SPLINE
SPL {X  -117.172, Y  +273.562, Z    +0.000, E1   -47.526, E3 -228450.483}
SPL {X  -141.985, Y  +308.763, Z    +0.000, E1   -38.695, E3 -228517.793}
SPL {X  -151.595, Y  +331.355, Z    +0.000, E1   -30.702, E3 -228532.311}
SPL {X  -155.358, Y  +344.279, Z    +0.000, E1   -24.937, E3 -228537.500}
SPL {X  -158.582, Y  +361.322, Z    +0.000, E1   -15.773, E3 -228541.844}
SPL {X  -159.657, Y  +372.183, Z    +0.000, E1    -8.995, E3 -228543.452}
SPL {X  -159.949, Y  +378.873, Z    +0.000, E1    -4.398, E3 -228544.026}
SPL {X  -159.990, Y  +382.801, Z    +0.000, E1    -1.461, E3 -228544.200}
SPL {X  -159.990, Y  +385.055, Z    +0.000, E1    +0.429, E3 -228544.239}
SPL {X  -159.990, Y  +388.743, Z    +0.000, E1    +5.147, E3 -228544.380}
SPL {X  -159.990, Y  +393.154, Z    +0.000, E1   +11.942, E3 -228544.712}
SPL {X  -159.990, Y  +397.198, Z    +0.000, E1   +18.490, E3 -228545.209}
SPL {X  -159.990, Y  +402.771, Z    +0.000, E1   +27.045, E3 -228546.172}
SPL {X  -159.990, Y  +416.096, Z    +0.000, E1   +42.325, E3 -228549.839}
SPL {X  -159.990, Y  +469.763, Z    +0.000, E1   +60.937, E3 -228575.069}
SPL {X  -159.990, Y  +561.242, Z    +0.000, E1   +63.988, E3 -228646.017}
SPL {X  -159.990, Y  +574.019, Z    +0.000, E1   +64.020, E3 -228659.184}
SPL {X  -159.990, Y  +591.720, Z    +0.000, E1   +64.032, E3 -228677.482}
SPL {X  -159.990, Y  +605.088, Z    +0.000, E1   +63.988, E3 -228691.409}
SPL {X  -159.990, Y  +614.683, Z    +0.000, E1   +63.997, E3 -228701.304}
SPL {X  -159.990, Y  +629.274, Z    +0.000, E1   +64.033, E3 -228716.335}
SPL {X  -159.990, Y  +645.396, Z    +0.000, E1   +64.010, E3 -228733.066}
SPL {X  -159.990, Y  +656.294, Z    +0.000, E1   +63.988, E3 -228744.396}
SPL {X  -159.990, Y  +667.666, Z    +0.000, E1   +64.016, E3 -228756.087}
SPL {X  -159.767, Y  +679.937, Z    +0.000, E1   +63.968, E3 -228769.063}
SPL {X  -159.113, Y  +688.225, Z    +0.000, E1   +63.867, E3 -228778.341}
SPL {X  -158.361, Y  +694.273, Z    +0.000, E1   +63.762, E3 -228785.378}
SPL {X  -157.131, Y  +701.612, Z    +0.000, E1   +63.591, E3 -228794.251}
SPL {X  -154.918, Y  +711.464, Z    +0.000, E1   +63.294, E3 -228806.686}
SPL {X  -151.874, Y  +721.810, Z    +0.000, E1   +62.834, E3 -228820.493}
SPL {X  -148.087, Y  +732.056, Z    +0.000, E1   +62.252, E3 -228834.850}
SPL {X  -144.667, Y  +739.825, Z    +0.000, E1   +61.658, E3 -228846.239}
SPL {X  -142.263, Y  +744.698, Z    +0.000, E1   +61.245, E3 -228853.554}
SPL {X  -139.956, Y  +749.019, Z    +0.000, E1   +60.852, E3 -228860.132}
SPL {X  -136.617, Y  +754.762, Z    +0.000, E1   +60.296, E3 -228868.986}
SPL {X  -132.995, Y  +760.433, Z    +0.000, E1   +59.601, E3 -228877.950}
SPL {X  -109.949, Y  +787.724, Z    +0.000, E1   +51.944, E3 -228970.511}
ENDSPLINE

SPLINE
SPL {X  -129.366, Y  +765.635, Z    +0.000, E1   +44.361, E3 -229080.253}
SPL {X  -144.719, Y  +739.715, Z    +0.000, E1   +37.620, E3 -229107.101}
SPL {X  -154.606, Y  +712.654, Z    +0.000, E1   +26.872, E3 -229120.321}
SPL {X  -158.229, Y  +695.175, Z    +0.000, E1   +17.621, E3 -229124.807}
SPL {X  -159.735, Y  +680.532, Z    +0.000, E1    +8.352, E3 -229126.899}
SPL {X  -159.976, Y  +673.579, Z    +0.000, E1    +3.308, E3 -229127.393}
SPL {X  -159.990, Y  +669.438, Z    +0.000, E1    +0.061, E3 -229127.491}
SPL {X  -159.990, Y  +667.221, Z    +0.000, E1    -2.789, E3 -229127.534}
SPL {X  -159.990, Y  +663.611, Z    +0.000, E1    -7.967, E3 -229127.724}
SPL {X  -159.990, Y  +658.381, Z    +0.000, E1   -16.786, E3 -229128.205}
SPL {X  -159.990, Y  +651.878, Z    +0.000, E1   -27.298, E3 -229129.204}
SPL {X  -159.990, Y  +644.587, Z    +0.000, E1   -37.284, E3 -229130.787}
SPL {X  -159.990, Y  +633.621, Z    +0.000, E1   -47.309, E3 -229134.278}
SPL {X  -159.990, Y  +588.658, Z    +0.000, E1   -60.812, E3 -229156.598}
SPL {X  -159.990, Y  +495.038, Z    +0.000, E1   -63.580, E3 -229231.834}
SPL {X  -159.990, Y  +483.848, Z    +0.000, E1   -63.590, E3 -229243.619}
SPL {X  -159.990, Y  +471.874, Z    +0.000, E1   -63.586, E3 -229256.245}
SPL {X  -159.990, Y  +461.079, Z    +0.000, E1   -63.579, E3 -229267.653}
SPL {X  -159.990, Y  +450.188, Z    +0.000, E1   -63.581, E3 -229279.144}
SPL {X  -159.990, Y  +442.553, Z    +0.000, E1   -63.337, E3 -229288.967}
ENDSPLINE

SPLINE
SPL {X  -159.990, Y  +465.419, Z    +0.000, E1   -58.181, E3 -229297.813}
ENDSPLINE

SPLINE
SPL {X  -159.990, Y  +455.003, Z    +0.000, E1   -58.788, E3 -229307.351}
SPL {X  -159.990, Y  +443.180, Z    +0.000, E1   -59.522, E3 -229317.389}
SPL {X  -159.990, Y  +431.227, Z    +0.000, E1   -60.120, E3 -229328.081}
SPL {X  -159.990, Y  +413.464, Z    +0.000, E1   -61.043, E3 -229343.071}
SPL {X  -159.990, Y  +395.417, Z    +0.000, E1   -62.063, E3 -229356.514}
SPL {X  -159.983, Y  +381.042, Z    +0.000, E1   -62.802, E3 -229367.145}
SPL {X  -159.542, Y  +370.537, Z    +0.000, E1   -63.069, E3 -229376.527}
SPL {X  -158.758, Y  +362.683, Z    +0.000, E1   -62.956, E3 -229385.801}
SPL {X  -157.125, Y  +352.357, Z    +0.000, E1   -62.751, E3 -229398.534}
SPL {X  -154.421, Y  +340.656, Z    +0.000, E1   -62.344, E3 -229413.888}
SPL {X  -151.938, Y  +332.383, Z    +0.000, E1   -61.927, E3 -229425.360}
SPL {X  -149.604, Y  +325.796, Z    +0.000, E1   -61.568, E3 -229434.746}
SPL {X  -147.413, Y  +320.320, Z    +0.000, E1   -61.198, E3 -229442.799}
SPL {X  -145.235, Y  +315.391, Z    +0.000, E1   -60.847, E3 -229450.174}
SPL {X  -141.610, Y  +308.046, Z    +0.000, E1   -60.266, E3 -229461.410}
SPL {X  -138.010, Y  +301.568, Z    +0.000, E1   -59.585, E3 -229471.682}
SPL {X  -134.495, Y  +295.853, Z    +0.000, E1   -58.965, E3 -229480.819}
SPL {X  -113.541, Y  +269.782, Z    +0.000, E1   -50.113, E3 -229588.412}
ENDSPLINE

SPLINE
SPL {X  -145.506, Y  +315.982, Z    +0.000, E1   -36.457, E3 -229701.647}
SPL {X  -155.358, Y  +344.279, Z    +0.000, E1   -24.937, E3 -229716.071}
SPL {X  -158.582, Y  +361.322, Z    +0.000, E1   -15.773, E3 -229720.415}
SPL {X  -159.657, Y  +372.183, Z    +0.000, E1    -8.995, E3 -229722.023}
SPL {X  -159.986, Y  +381.348, Z    +0.000, E1    -2.678, E3 -229722.712}
SPL {X  -159.990, Y  +385.055, Z    +0.000, E1    +0.429, E3 -229722.811}
SPL {X  -159.990, Y  +388.743, Z    +0.000, E1    +5.147, E3 -229722.951}
SPL {X  -159.990, Y  +393.154, Z    +0.000, E1   +11.942, E3 -229723.283}
SPL {X  -159.990, Y  +397.198, Z    +0.000, E1   +18.490, E3 -229723.780}
SPL {X  -159.990, Y  +402.771, Z    +0.000, E1   +27.045, E3 -229724.743}
SPL {X  -159.990, Y  +416.096, Z    +0.000, E1   +42.325, E3 -229728.411}
SPL {X  -159.990, Y  +469.763, Z    +0.000, E1   +60.937, E3 -229753.641}
SPL {X  -159.990, Y  +565.969, Z    +0.000, E1   +64.023, E3 -229829.414}
SPL {X  -159.990, Y  +578.082, Z    +0.000, E1   +63.987, E3 -229842.023}
SPL {X  -159.990, Y  +588.139, Z    +0.000, E1   +64.000, E3 -229852.403}
SPL {X  -159.990, Y  +601.786, Z    +0.000, E1   +64.016, E3 -229866.507}
SPL {X  -159.990, Y  +614.683, Z    +0.000, E1   +63.997, E3 -229879.875}
SPL {X  -159.990, Y  +629.274, Z    +0.000, E1   +64.033, E3 -229894.906}
SPL {X  -159.990, Y  +645.396, Z    +0.000, E1   +64.010, E3 -229911.637}
SPL {X  -159.990, Y  +656.294, Z    +0.000, E1   +63.988, E3 -229922.967}
SPL {X  -159.990, Y  +667.666, Z    +0.000, E1   +64.016, E3 -229934.659}
SPL {X  -159.767, Y  +679.937, Z    +0.000, E1   +63.968, E3 -229947.634}
SPL {X  -158.736, Y  +691.491, Z    +0.000, E1   +63.843, E3 -229960.633}
SPL {X  -157.131, Y  +701.612, Z    +0.000, E1   +63.591, E3 -229972.823}
SPL {X  -154.918, Y  +711.464, Z    +0.000, E1   +63.294, E3 -229985.258}
SPL {X  -152.656, Y  +719.385, Z    +0.000, E1   +62.921, E3 -229995.826}
SPL {X  -150.233, Y  +726.516, Z    +0.000, E1   +62.565, E3 -230005.604}
SPL {X  -147.385, Y  +733.745, Z    +0.000, E1   +62.104, E3 -230015.908}
SPL {X  -144.667, Y  +739.825, Z    +0.000, E1   +61.658, E3 -230024.811}
SPL {X  -142.263, Y  +744.698, Z    +0.000, E1   +61.245, E3 -230032.126}
SPL {X  -139.956, Y  +749.019, Z    +0.000, E1   +60.852, E3 -230038.703}
SPL {X  -136.617, Y  +754.762, Z    +0.000, E1   +60.296, E3 -230047.557}
SPL {X  -132.995, Y  +760.433, Z    +0.000, E1   +59.601, E3 -230056.521}
SPL {X  -109.949, Y  +787.724, Z    +0.000, E1   +51.944, E3 -230149.083}
ENDSPLINE

SPLINE
SPL {X  -129.366, Y  +765.635, Z    +0.000, E1   +44.361, E3 -230258.825}
SPL {X  -144.719, Y  +739.715, Z    +0.000, E1   +37.620, E3 -230285.672}
SPL {X  -154.606, Y  +712.654, Z    +0.000, E1   +26.872, E3 -230298.892}
SPL {X  -158.229, Y  +695.175, Z    +0.000, E1   +17.621, E3 -230303.378}
SPL {X  -159.735, Y  +680.532, Z    +0.000, E1    +8.352, E3 -230305.470}
SPL {X  -159.990, Y  +671.731, Z    +0.000, E1    +1.953, E3 -230306.020}
SPL {X  -159.990, Y  +669.188, Z    +0.000, E1    -0.261, E3 -230306.065}
SPL {X  -159.990, Y  +666.135, Z    +0.000, E1    -4.178, E3 -230306.154}
SPL {X  -159.990, Y  +662.249, Z    +0.000, E1   -10.338, E3 -230306.385}
SPL {X  -159.990, Y  +658.381, Z    +0.000, E1   -16.786, E3 -230306.777}
SPL {X  -159.990, Y  +651.878, Z    +0.000, E1   -27.298, E3 -230307.776}
SPL {X  -159.990, Y  +644.587, Z    +0.000, E1   -37.284, E3 -230309.358}
SPL {X  -159.990, Y  +633.621, Z    +0.000, E1   -47.309, E3 -230312.849}
SPL {X  -159.990, Y  +588.658, Z    +0.000, E1   -60.812, E3 -230335.169}
SPL {X  -159.990, Y  +495.038, Z    +0.000, E1   -63.580, E3 -230410.406}
SPL {X  -159.990, Y  +483.848, Z    +0.000, E1   -63.590, E3 -230422.190}
SPL {X  -159.990, Y  +471.874, Z    +0.000, E1   -63.586, E3 -230434.816}
SPL {X  -159.990, Y  +461.079, Z    +0.000, E1   -63.579, E3 -230446.225}
SPL {X  -159.990, Y  +450.188, Z    +0.000, E1   -63.581, E3 -230457.715}
SPL {X  -159.990, Y  +442.553, Z    +0.000, E1   -63.337, E3 -230467.539}
ENDSPLINE

SPLINE
SPL {X  -159.990, Y  +465.419, Z    +0.000, E1   -58.181, E3 -230476.384}
ENDSPLINE

SPLINE
SPL {X  -159.990, Y  +455.003, Z    +0.000, E1   -58.788, E3 -230485.922}
SPL {X  -159.990, Y  +443.180, Z    +0.000, E1   -59.522, E3 -230495.961}
SPL {X  -159.990, Y  +431.227, Z    +0.000, E1   -60.120, E3 -230506.653}
SPL {X  -159.990, Y  +413.464, Z    +0.000, E1   -61.043, E3 -230521.643}
SPL {X  -159.990, Y  +395.417, Z    +0.000, E1   -62.063, E3 -230535.086}
SPL {X  -159.983, Y  +381.042, Z    +0.000, E1   -62.802, E3 -230545.717}
SPL {X  -159.542, Y  +370.537, Z    +0.000, E1   -63.069, E3 -230555.099}
SPL {X  -158.758, Y  +362.683, Z    +0.000, E1   -62.956, E3 -230564.373}
SPL {X  -157.125, Y  +352.357, Z    +0.000, E1   -62.751, E3 -230577.106}
SPL {X  -154.421, Y  +340.656, Z    +0.000, E1   -62.344, E3 -230592.459}
SPL {X  -151.938, Y  +332.383, Z    +0.000, E1   -61.927, E3 -230603.932}
SPL {X  -149.604, Y  +325.796, Z    +0.000, E1   -61.568, E3 -230613.318}
SPL {X  -147.413, Y  +320.320, Z    +0.000, E1   -61.198, E3 -230621.371}
SPL {X  -145.235, Y  +315.391, Z    +0.000, E1   -60.847, E3 -230628.746}
SPL {X  -141.610, Y  +308.046, Z    +0.000, E1   -60.266, E3 -230639.982}
SPL {X  -138.010, Y  +301.568, Z    +0.000, E1   -59.585, E3 -230650.253}
SPL {X  -134.495, Y  +295.853, Z    +0.000, E1   -58.965, E3 -230659.391}
SPL {X  -113.541, Y  +269.782, Z    +0.000, E1   -50.113, E3 -230766.983}
ENDSPLINE

SPLINE
SPL {X  -141.985, Y  +308.763, Z    +0.000, E1   -38.695, E3 -230874.935}
SPL {X  -154.491, Y  +340.913, Z    +0.000, E1   -26.570, E3 -230893.388}
SPL {X  -158.582, Y  +361.322, Z    +0.000, E1   -15.773, E3 -230898.987}
SPL {X  -159.657, Y  +372.183, Z    +0.000, E1    -8.995, E3 -230900.595}
SPL {X  -159.986, Y  +381.348, Z    +0.000, E1    -2.678, E3 -230901.283}
SPL {X  -159.990, Y  +384.517, Z    +0.000, E1    -0.022, E3 -230901.373}
SPL {X  -159.990, Y  +386.497, Z    +0.000, E1    +2.123, E3 -230901.421}
SPL {X  -159.990, Y  +391.572, Z    +0.000, E1    +9.236, E3 -230901.727}
SPL {X  -159.990, Y  +397.198, Z    +0.000, E1   +18.490, E3 -230902.352}
SPL {X  -159.990, Y  +402.771, Z    +0.000, E1   +27.045, E3 -230903.315}
SPL {X  -159.990, Y  +416.096, Z    +0.000, E1   +42.325, E3 -230906.982}
SPL {X  -159.990, Y  +469.763, Z    +0.000, E1   +60.937, E3 -230932.212}
SPL {X  -159.990, Y  +561.242, Z    +0.000, E1   +63.988, E3 -231003.160}
SPL {X  -159.990, Y  +574.019, Z    +0.000, E1   +64.020, E3 -231016.326}
SPL {X  -159.990, Y  +591.720, Z    +0.000, E1   +64.032, E3 -231034.625}
SPL {X  -159.990, Y  +605.088, Z    +0.000, E1   +63.988, E3 -231048.552}
SPL {X  -159.990, Y  +614.683, Z    +0.000, E1   +63.997, E3 -231058.447}
SPL {X  -159.990, Y  +629.274, Z    +0.000, E1   +64.033, E3 -231073.478}
SPL {X  -159.990, Y  +645.396, Z    +0.000, E1   +64.010, E3 -231090.209}
SPL {X  -159.990, Y  +656.294, Z    +0.000, E1   +63.988, E3 -231101.539}
SPL {X  -159.990, Y  +667.666, Z    +0.000, E1   +64.016, E3 -231113.230}
SPL {X  -159.767, Y  +679.937, Z    +0.000, E1   +63.968, E3 -231126.206}
SPL {X  -159.113, Y  +688.225, Z    +0.000, E1   +63.867, E3 -231135.483}
SPL {X  -158.361, Y  +694.273, Z    +0.000, E1   +63.762, E3 -231142.521}
SPL {X  -157.131, Y  +701.612, Z    +0.000, E1   +63.591, E3 -231151.394}
SPL {X  -154.918, Y  +711.464, Z    +0.000, E1   +63.294, E3 -231163.829}
SPL {X  -151.874, Y  +721.810, Z    +0.000, E1   +62.834, E3 -231177.636}
SPL {X  -148.087, Y  +732.056, Z    +0.000, E1   +62.252, E3 -231191.993}
SPL {X  -144.667, Y  +739.825, Z    +0.000, E1   +61.658, E3 -231203.382}
SPL {X  -142.263, Y  +744.698, Z    +0.000, E1   +61.245, E3 -231210.697}
SPL {X  -138.935, Y  +750.833, Z    +0.000, E1   +60.711, E3 -231220.022}
SPL {X  -135.668, Y  +756.300, Z    +0.000, E1   +60.086, E3 -231228.585}
SPL {X  -132.995, Y  +760.433, Z    +0.000, E1   +59.601, E3 -231235.093}
SPL {X  -109.949, Y  +787.724, Z    +0.000, E1   +51.944, E3 -231327.654}
ENDSPLINE

SPLINE
SPL {X  -129.366, Y  +765.635, Z    +0.000, E1   +44.361, E3 -231437.396}
SPL {X  -144.719, Y  +739.715, Z    +0.000, E1   +37.620, E3 -231464.244}
SPL {X  -154.606, Y  +712.654, Z    +0.000, E1   +26.872, E3 -231477.464}
SPL {X  -158.229, Y  +695.175, Z    +0.000, E1   +17.621, E3 -231481.950}
SPL {X  -159.735, Y  +680.532, Z    +0.000, E1    +8.352, E3 -231484.042}
SPL {X  -159.990, Y  +671.731, Z    +0.000, E1    +1.953, E3 -231484.592}
SPL {X  -159.990, Y  +669.188, Z    +0.000, E1    -0.261, E3 -231484.636}
SPL {X  -159.990, Y  +666.135, Z    +0.000, E1    -4.178, E3 -231484.725}
SPL {X  -159.990, Y  +662.249, Z    +0.000, E1   -10.338, E3 -231484.956}
SPL {X  -159.990, Y  +658.381, Z    +0.000, E1   -16.786, E3 -231485.348}
SPL {X  -159.990, Y  +651.878, Z    +0.000, E1   -27.298, E3 -231486.347}
SPL {X  -159.990, Y  +644.587, Z    +0.000, E1   -37.284, E3 -231487.930}
SPL {X  -159.990, Y  +633.621, Z    +0.000, E1   -47.309, E3 -231491.421}
SPL {X  -159.990, Y  +588.658, Z    +0.000, E1   -60.812, E3 -231513.741}
SPL {X  -159.990, Y  +495.038, Z    +0.000, E1   -63.580, E3 -231588.977}
SPL {X  -159.990, Y  +483.848, Z    +0.000, E1   -63.590, E3 -231600.762}
SPL {X  -159.990, Y  +471.874, Z    +0.000, E1   -63.586, E3 -231613.387}
SPL {X  -159.990, Y  +461.079, Z    +0.000, E1   -63.579, E3 -231624.796}
SPL {X  -159.990, Y  +450.188, Z    +0.000, E1   -63.581, E3 -231636.287}
SPL {X  -159.990, Y  +442.553, Z    +0.000, E1   -63.337, E3 -231646.110}
ENDSPLINE

SPLINE
SPL {X  -159.990, Y  +465.419, Z    +0.000, E1   -58.181, E3 -231654.956}
ENDSPLINE

SPLINE
SPL {X  -159.990, Y  +455.003, Z    +0.000, E1   -58.788, E3 -231664.494}
SPL {X  -159.990, Y  +443.180, Z    +0.000, E1   -59.522, E3 -231674.532}
SPL {X  -159.990, Y  +431.227, Z    +0.000, E1   -60.120, E3 -231685.224}
SPL {X  -159.990, Y  +413.464, Z    +0.000, E1   -61.043, E3 -231700.214}
SPL {X  -159.990, Y  +395.417, Z    +0.000, E1   -62.063, E3 -231713.657}
SPL {X  -159.982, Y  +380.853, Z    +0.000, E1   -62.802, E3 -231724.504}
ENDSPLINE

SPLINE
SPL {X  -159.990, Y  +396.036, Z    +0.000, E1   -58.804, E3 -231734.138}
ENDSPLINE

SPLINE
SPL {X  -159.990, Y  +387.403, Z    +0.000, E1   -58.805, E3 -231745.251}
SPL {X  -159.948, Y  +378.844, Z    +0.000, E1   -58.798, E3 -231756.291}
SPL {X  -159.570, Y  +370.916, Z    +0.000, E1   -58.738, E3 -231766.887}
SPL {X  -158.865, Y  +363.563, Z    +0.000, E1   -58.615, E3 -231777.096}
SPL {X  -157.976, Y  +357.197, Z    +0.000, E1   -58.476, E3 -231786.197}
SPL {X  -156.730, Y  +350.368, Z    +0.000, E1   -58.276, E3 -231796.292}
SPL {X  -155.026, Y  +342.956, Z    +0.000, E1   -58.003, E3 -231807.564}
SPL {X  -152.946, Y  +335.551, Z    +0.000, E1   -57.653, E3 -231819.212}
SPL {X  -150.899, Y  +329.336, Z    +0.000, E1   -57.290, E3 -231829.278}
SPL {X  -149.179, Y  +324.687, Z    +0.000, E1   -56.983, E3 -231836.967}
SPL {X  -147.281, Y  +320.009, Z    +0.000, E1   -56.662, E3 -231844.793}
SPL {X  -144.114, Y  +313.017, Z    +0.000, E1   -56.131, E3 -231856.761}
SPL {X  -140.858, Y  +306.633, Z    +0.000, E1   -55.477, E3 -231868.056}
SPL {X  -138.338, Y  +302.130, Z    +0.000, E1   -54.992, E3 -231876.106}
SPL {X  -124.427, Y  +281.929, Z    +0.000, E1   -46.852, E3 -231980.342}
ENDSPLINE

SPLINE
SPL {X  -148.251, Y  +322.346, Z    +0.000, E1   -33.039, E3 -232068.267}
SPL {X  -157.534, Y  +354.574, Z    +0.000, E1   -18.815, E3 -232085.096}
SPL {X  -159.548, Y  +370.614, Z    +0.000, E1    -9.656, E3 -232088.721}
SPL {X  -159.928, Y  +378.035, Z    +0.000, E1    -4.866, E3 -232089.637}
SPL {X  -159.990, Y  +383.381, Z    +0.000, E1    -1.123, E3 -232089.958}
SPL {X  -159.990, Y  +385.440, Z    +0.000, E1    +0.747, E3 -232090.027}
SPL {X  -159.990, Y  +388.179, Z    +0.000, E1    +3.660, E3 -232090.168}
SPL {X  -159.990, Y  +394.222, Z    +0.000, E1   +11.674, E3 -232090.761}
SPL {X  -159.990, Y  +403.976, Z    +0.000, E1   +25.456, E3 -232092.640}
SPL {X  -159.990, Y  +417.120, Z    +0.000, E1   +39.678, E3 -232096.672}
SPL {X  -159.990, Y  +456.927, Z    +0.000, E1   +55.382, E3 -232118.532}
SPL {X  -159.990, Y  +530.047, Z    +0.000, E1   +58.901, E3 -232188.366}
SPL {X  -159.990, Y  +538.035, Z    +0.000, E1   +58.900, E3 -232198.591}
SPL {X  -159.990, Y  +546.883, Z    +0.000, E1   +58.912, E3 -232209.895}
SPL {X  -159.990, Y  +555.949, Z    +0.000, E1   +58.900, E3 -232221.514}
SPL {X  -159.990, Y  +563.718, Z    +0.000, E1   +58.903, E3 -232231.435}
SPL {X  -159.990, Y  +571.529, Z    +0.000, E1   +58.906, E3 -232241.419}
SPL {X  -159.990, Y  +579.859, Z    +0.000, E1   +58.907, E3 -232252.078}
SPL {X  -159.990, Y  +588.526, Z    +0.000, E1   +58.910, E3 -232263.152}
SPL {X  -159.990, Y  +596.521, Z    +0.000, E1   +58.902, E3 -232273.411}
SPL {X  -159.990, Y  +605.444, Z    +0.000, E1   +58.918, E3 -232284.800}
SPL {X  -159.990, Y  +618.101, Z    +0.000, E1   +58.946, E3 -232300.947}
SPL {X  -159.990, Y  +629.920, Z    +0.000, E1   +58.912, E3 -232316.140}
SPL {X  -159.990, Y  +638.424, Z    +0.000, E1   +58.901, E3 -232327.040}
SPL {X  -159.990, Y  +645.995, Z    +0.000, E1   +58.900, E3 -232336.728}
SPL {X  -159.990, Y  +654.206, Z    +0.000, E1   +58.908, E3 -232347.218}
SPL {X  -159.990, Y  +661.562, Z    +0.000, E1   +58.900, E3 -232356.647}
SPL {X  -159.990, Y  +670.328, Z    +0.000, E1   +58.911, E3 -232367.846}
SPL {X  -159.795, Y  +679.404, Z    +0.000, E1   +58.876, E3 -232379.671}
SPL {X  -159.282, Y  +686.534, Z    +0.000, E1   +58.787, E3 -232389.345}
SPL {X  -158.463, Y  +693.553, Z    +0.000, E1   +58.665, E3 -232399.186}
SPL {X  -157.294, Y  +700.745, Z    +0.000, E1   +58.469, E3 -232409.636}
SPL {X  -156.031, Y  +706.871, Z    +0.000, E1   +58.260, E3 -232418.782}
SPL {X  -154.558, Y  +712.835, Z    +0.000, E1   +58.028, E3 -232427.909}
SPL {X  -152.750, Y  +719.085, Z    +0.000, E1   +57.721, E3 -232437.755}
SPL {X  -150.741, Y  +725.111, Z    +0.000, E1   +57.387, E3 -232447.459}
SPL {X  -148.665, Y  +730.623, Z    +0.000, E1   +57.007, E3 -232456.608}
SPL {X  -146.664, Y  +735.425, Z    +0.000, E1   +56.657, E3 -232464.698}
SPL {X  -144.631, Y  +739.900, Z    +0.000, E1   +56.280, E3 -232472.383}
SPL {X  -141.795, Y  +745.600, Z    +0.000, E1   +55.801, E3 -232482.266}
SPL {X  -138.492, Y  +751.605, Z    +0.000, E1   +55.137, E3 -232492.990}
SPL {X  -124.324, Y  +772.199, Z    +0.000, E1   +48.708, E3 -232571.998}
ENDSPLINE

SPLINE
SPL {X  -129.118, Y  +765.975, Z    +0.000, E1   +43.713, E3 -232636.483}
SPL {X  -146.252, Y  +736.362, Z    +0.000, E1   +34.795, E3 -232685.661}
SPL {X  -155.916, Y  +707.374, Z    +0.000, E1   +22.878, E3 -232702.546}
SPL {X  -159.039, Y  +688.920, Z    +0.000, E1   +13.016, E3 -232707.781}
SPL {X  -159.777, Y  +679.762, Z    +0.000, E1    +7.372, E3 -232709.236}
SPL {X  -159.984, Y  +672.872, Z    +0.000, E1    +2.784, E3 -232709.833}
SPL {X  -159.990, Y  +668.898, Z    +0.000, E1    -0.346, E3 -232709.991}
SPL {X  -159.990, Y  +666.084, Z    +0.000, E1    -3.512, E3 -232710.114}
SPL {X  -159.990, Y  +662.904, Z    +0.000, E1    -7.618, E3 -232710.353}
SPL {X  -159.990, Y  +658.509, Z    +0.000, E1   -13.882, E3 -232710.889}
SPL {X  -159.990, Y  +652.317, Z    +0.000, E1   -22.778, E3 -232712.024}
SPL {X  -159.990, Y  +640.689, Z    +0.000, E1   -37.390, E3 -232713.567}
SPL {X  -159.990, Y  +585.634, Z    +0.000, E1   -68.681, E3 -232714.191}
SPL {X  -159.990, Y  +457.771, Z    +0.000, E1   -68.079, E3 -232804.752}
SPL {X  -159.990, Y  +453.218, Z    +0.000, E1   -67.322, E3 -232815.188}
SPL {X  -159.990, Y  +450.256, Z    +0.000, E1   -66.188, E3 -232827.120}
SPL {X  -159.990, Y  +445.667, Z    +0.000, E1   -65.356, E3 -232838.032}
SPL {X  -159.990, Y  +439.738, Z    +0.000, E1   -64.716, E3 -232848.845}
SPL {X  -159.990, Y  +435.528, Z    +0.000, E1   -63.972, E3 -232858.721}
SPL {X  -159.990, Y  +429.021, Z    +0.000, E1   -63.228, E3 -232871.333}
SPL {X  -159.990, Y  +423.267, Z    +0.000, E1   -62.365, E3 -232883.631}
SPL {X  -159.990, Y  +418.218, Z    +0.000, E1   -61.769, E3 -232893.644}
SPL {X  -159.990, Y  +412.274, Z    +0.000, E1   -61.123, E3 -232905.048}
SPL {X  -159.990, Y  +408.631, Z    +0.000, E1   -60.233, E3 -232915.510}
SPL {X  -159.990, Y  +402.821, Z    +0.000, E1   -59.334, E3 -232929.037}
SPL {X  -159.990, Y  +395.849, Z    +0.000, E1   -58.799, E3 -232941.302}
SPL {X  -159.990, Y  +387.403, Z    +0.000, E1   -58.805, E3 -232952.148}
SPL {X  -159.948, Y  +378.844, Z    +0.000, E1   -58.798, E3 -232963.188}
SPL {X  -159.570, Y  +370.916, Z    +0.000, E1   -58.738, E3 -232973.783}
SPL {X  -158.865, Y  +363.563, Z    +0.000, E1   -58.615, E3 -232983.992}
SPL {X  -157.976, Y  +357.197, Z    +0.000, E1   -58.476, E3 -232993.093}
SPL {X  -156.730, Y  +350.368, Z    +0.000, E1   -58.276, E3 -233003.189}
SPL {X  -155.026, Y  +342.956, Z    +0.000, E1   -58.003, E3 -233014.461}
SPL {X  -152.946, Y  +335.551, Z    +0.000, E1   -57.653, E3 -233026.109}
SPL {X  -150.105, Y  +327.135, Z    +0.000, E1   -57.196, E3 -233039.729}
SPL {X  -147.281, Y  +320.009, Z    +0.000, E1   -56.662, E3 -233051.690}
SPL {X  -144.114, Y  +313.017, Z    +0.000, E1   -56.131, E3 -233063.657}
SPL {X  -140.858, Y  +306.633, Z    +0.000, E1   -55.477, E3 -233074.953}
SPL {X  -138.338, Y  +302.130, Z    +0.000, E1   -54.992, E3 -233083.002}
SPL {X  -124.427, Y  +281.929, Z    +0.000, E1   -46.852, E3 -233187.238}
ENDSPLINE

SPLINE
SPL {X  -148.251, Y  +322.346, Z    +0.000, E1   -33.039, E3 -233275.164}
SPL {X  -157.534, Y  +354.574, Z    +0.000, E1   -18.815, E3 -233291.993}
SPL {X  -159.548, Y  +370.614, Z    +0.000, E1    -9.656, E3 -233295.618}
SPL {X  -159.973, Y  +380.173, Z    +0.000, E1    -3.469, E3 -233296.685}
SPL {X  -159.990, Y  +384.791, Z    +0.000, E1    +0.055, E3 -233296.904}
SPL {X  -159.990, Y  +388.179, Z    +0.000, E1    +3.660, E3 -233297.064}
SPL {X  -159.990, Y  +394.222, Z    +0.000, E1   +11.674, E3 -233297.657}
SPL {X  -159.990, Y  +403.976, Z    +0.000, E1   +25.456, E3 -233299.537}
SPL {X  -159.990, Y  +417.120, Z    +0.000, E1   +39.678, E3 -233303.568}
SPL {X  -159.990, Y  +456.927, Z    +0.000, E1   +55.382, E3 -233325.429}
SPL {X  -159.990, Y  +530.047, Z    +0.000, E1   +58.901, E3 -233395.263}
SPL {X  -159.990, Y  +538.035, Z    +0.000, E1   +58.900, E3 -233405.488}
SPL {X  -159.990, Y  +546.883, Z    +0.000, E1   +58.912, E3 -233416.792}
SPL {X  -159.990, Y  +555.949, Z    +0.000, E1   +58.900, E3 -233428.411}
SPL {X  -159.990, Y  +563.718, Z    +0.000, E1   +58.903, E3 -233438.331}
SPL {X  -159.990, Y  +571.529, Z    +0.000, E1   +58.906, E3 -233448.315}
SPL {X  -159.990, Y  +579.859, Z    +0.000, E1   +58.907, E3 -233458.975}
SPL {X  -159.990, Y  +588.526, Z    +0.000, E1   +58.910, E3 -233470.048}
SPL {X  -159.990, Y  +596.521, Z    +0.000, E1   +58.902, E3 -233480.307}
SPL {X  -159.990, Y  +605.444, Z    +0.000, E1   +58.918, E3 -233491.697}
SPL {X  -159.990, Y  +613.908, Z    +0.000, E1   +58.900, E3 -233502.556}
SPL {X  -159.990, Y  +621.342, Z    +0.000, E1   +58.904, E3 -233512.064}
SPL {X  -159.990, Y  +629.920, Z    +0.000, E1   +58.912, E3 -233523.037}
SPL {X  -159.990, Y  +642.398, Z    +0.000, E1   +58.947, E3 -233538.944}
SPL {X  -159.990, Y  +654.206, Z    +0.000, E1   +58.908, E3 -233554.115}
SPL {X  -159.990, Y  +661.562, Z    +0.000, E1   +58.900, E3 -233563.543}
SPL {X  -159.990, Y  +670.328, Z    +0.000, E1   +58.911, E3 -233574.742}
SPL {X  -159.795, Y  +679.404, Z    +0.000, E1   +58.876, E3 -233586.568}
SPL {X  -159.282, Y  +686.534, Z    +0.000, E1   +58.787, E3 -233596.241}
SPL {X  -158.463, Y  +693.553, Z    +0.000, E1   +58.665, E3 -233606.083}
SPL {X  -157.294, Y  +700.745, Z    +0.000, E1   +58.469, E3 -233616.533}
SPL {X  -156.031, Y  +706.871, Z    +0.000, E1   +58.260, E3 -233625.678}
SPL {X  -154.558, Y  +712.835, Z    +0.000, E1   +58.028, E3 -233634.805}
SPL {X  -152.750, Y  +719.085, Z    +0.000, E1   +57.721, E3 -233644.652}
SPL {X  -150.741, Y  +725.111, Z    +0.000, E1   +57.387, E3 -233654.356}
SPL {X  -148.665, Y  +730.623, Z    +0.000, E1   +57.007, E3 -233663.504}
SPL {X  -146.664, Y  +735.425, Z    +0.000, E1   +56.657, E3 -233671.594}
SPL {X  -143.496, Y  +742.251, Z    +0.000, E1   +56.124, E3 -233683.288}
SPL {X  -140.752, Y  +747.564, Z    +0.000, E1   +55.554, E3 -233692.695}
SPL {X  -138.492, Y  +751.605, Z    +0.000, E1   +55.137, E3 -233699.886}
SPL {X  -124.324, Y  +772.199, Z    +0.000, E1   +48.708, E3 -233778.894}
ENDSPLINE

SPLINE
SPL {X  -129.118, Y  +765.975, Z    +0.000, E1   +43.713, E3 -233843.380}
SPL {X  -146.252, Y  +736.362, Z    +0.000, E1   +34.795, E3 -233892.557}
SPL {X  -154.088, Y  +714.555, Z    +0.000, E1   +26.177, E3 -233906.574}
SPL {X  -156.688, Y  +703.837, Z    +0.000, E1   +21.096, E3 -233910.745}
SPL {X  -159.039, Y  +688.920, Z    +0.000, E1   +13.016, E3 -233914.677}
SPL {X  -159.888, Y  +677.224, Z    +0.000, E1    +5.773, E3 -233916.390}
SPL {X  -159.990, Y  +670.275, Z    +0.000, E1    +0.854, E3 -233916.844}
SPL {X  -159.990, Y  +667.097, Z    +0.000, E1    -2.190, E3 -233916.961}
SPL {X  -159.990, Y  +662.904, Z    +0.000, E1    -7.618, E3 -233917.250}
SPL {X  -159.990, Y  +658.509, Z    +0.000, E1   -13.882, E3 -233917.785}
SPL {X  -159.990, Y  +652.317, Z    +0.000, E1   -22.778, E3 -233918.921}
SPL {X  -159.990, Y  +640.689, Z    +0.000, E1   -37.390, E3 -233920.463}
SPL {X  -159.990, Y  +585.634, Z    +0.000, E1   -68.681, E3 -233921.088}
SPL {X  -159.990, Y  +457.771, Z    +0.000, E1   -68.079, E3 -234011.649}
SPL {X  -159.990, Y  +453.218, Z    +0.000, E1   -67.322, E3 -234022.084}
SPL {X  -159.990, Y  +450.256, Z    +0.000, E1   -66.188, E3 -234034.017}
SPL {X  -159.990, Y  +445.667, Z    +0.000, E1   -65.356, E3 -234044.929}
SPL {X  -159.990, Y  +439.738, Z    +0.000, E1   -64.716, E3 -234055.741}
SPL {X  -159.990, Y  +435.528, Z    +0.000, E1   -63.972, E3 -234065.617}
SPL {X  -159.990, Y  +429.021, Z    +0.000, E1   -63.228, E3 -234078.230}
SPL {X  -159.990, Y  +423.267, Z    +0.000, E1   -62.365, E3 -234090.528}
SPL {X  -159.990, Y  +418.218, Z    +0.000, E1   -61.769, E3 -234100.540}
SPL {X  -159.990, Y  +412.274, Z    +0.000, E1   -61.123, E3 -234111.944}
SPL {X  -159.990, Y  +408.631, Z    +0.000, E1   -60.233, E3 -234122.407}
SPL {X  -159.990, Y  +402.821, Z    +0.000, E1   -59.334, E3 -234135.934}
SPL {X  -159.990, Y  +395.849, Z    +0.000, E1   -58.799, E3 -234148.198}
SPL {X  -159.990, Y  +387.403, Z    +0.000, E1   -58.805, E3 -234159.044}
SPL {X  -159.948, Y  +378.844, Z    +0.000, E1   -58.798, E3 -234170.084}
SPL {X  -159.570, Y  +370.916, Z    +0.000, E1   -58.738, E3 -234180.680}
SPL {X  -158.865, Y  +363.563, Z    +0.000, E1   -58.615, E3 -234190.889}
SPL {X  -157.976, Y  +357.197, Z    +0.000, E1   -58.476, E3 -234199.990}
SPL {X  -156.730, Y  +350.368, Z    +0.000, E1   -58.276, E3 -234210.085}
SPL {X  -155.026, Y  +342.956, Z    +0.000, E1   -58.003, E3 -234221.357}
SPL {X  -152.946, Y  +335.551, Z    +0.000, E1   -57.653, E3 -234233.005}
SPL {X  -150.105, Y  +327.135, Z    +0.000, E1   -57.196, E3 -234246.625}
SPL {X  -146.578, Y  +318.377, Z    +0.000, E1   -56.572, E3 -234261.318}
SPL {X  -143.463, Y  +311.683, Z    +0.000, E1   -55.972, E3 -234272.932}
SPL {X  -140.858, Y  +306.633, Z    +0.000, E1   -55.477, E3 -234281.849}
SPL {X  -138.338, Y  +302.130, Z    +0.000, E1   -54.992, E3 -234289.899}
SPL {X  -124.427, Y  +281.929, Z    +0.000, E1   -46.852, E3 -234394.135}
ENDSPLINE

SPLINE
SPL {X  -148.251, Y  +322.346, Z    +0.000, E1   -33.039, E3 -234482.060}
SPL {X  -157.534, Y  +354.574, Z    +0.000, E1   -18.815, E3 -234498.889}
SPL {X  -159.548, Y  +370.614, Z    +0.000, E1    -9.656, E3 -234502.514}
SPL {X  -159.973, Y  +380.173, Z    +0.000, E1    -3.469, E3 -234503.582}
SPL {X  -159.990, Y  +384.078, Z    +0.000, E1    -0.490, E3 -234503.779}
SPL {X  -159.990, Y  +386.348, Z    +0.000, E1    +1.571, E3 -234503.860}
SPL {X  -159.990, Y  +391.422, Z    +0.000, E1    +7.757, E3 -234504.234}
SPL {X  -159.990, Y  +399.099, Z    +0.000, E1   +18.787, E3 -234505.340}
SPL {X  -159.990, Y  +406.316, Z    +0.000, E1   +28.569, E3 -234507.018}
SPL {X  -159.990, Y  +417.120, Z    +0.000, E1   +39.678, E3 -234510.465}
SPL {X  -159.990, Y  +456.927, Z    +0.000, E1   +55.382, E3 -234532.325}
SPL {X  -159.990, Y  +530.047, Z    +0.000, E1   +58.901, E3 -234602.159}
SPL {X  -159.990, Y  +538.035, Z    +0.000, E1   +58.900, E3 -234612.384}
SPL {X  -159.990, Y  +546.883, Z    +0.000, E1   +58.912, E3 -234623.688}
SPL {X  -159.990, Y  +555.949, Z    +0.000, E1   +58.900, E3 -234635.308}
SPL {X  -159.990, Y  +563.718, Z    +0.000, E1   +58.903, E3 -234645.228}
SPL {X  -159.990, Y  +571.529, Z    +0.000, E1   +58.906, E3 -234655.212}
SPL {X  -159.990, Y  +579.859, Z    +0.000, E1   +58.907, E3 -234665.871}
SPL {X  -159.990, Y  +588.526, Z    +0.000, E1   +58.910, E3 -234676.945}
SPL {X  -159.990, Y  +596.521, Z    +0.000, E1   +58.902, E3 -234687.204}
SPL {X  -159.990, Y  +605.444, Z    +0.000, E1   +58.918, E3 -234698.593}
SPL {X  -159.990, Y  +613.908, Z    +0.000, E1   +58.900, E3 -234709.452}
SPL {X  -159.990, Y  +621.342, Z    +0.000, E1   +58.904, E3 -234718.961}
SPL {X  -159.990, Y  +629.920, Z    +0.000, E1   +58.912, E3 -234729.933}
SPL {X  -159.990, Y  +642.398, Z    +0.000, E1   +58.947, E3 -234745.841}
SPL {X  -159.990, Y  +654.206, Z    +0.000, E1   +58.908, E3 -234761.012}
SPL {X  -159.990, Y  +661.562, Z    +0.000, E1   +58.900, E3 -234770.440}
SPL {X  -159.990, Y  +670.328, Z    +0.000, E1   +58.911, E3 -234781.639}
SPL {X  -159.795, Y  +679.404, Z    +0.000, E1   +58.876, E3 -234793.464}
SPL {X  -159.282, Y  +686.534, Z    +0.000, E1   +58.787, E3 -234803.138}
SPL {X  -158.463, Y  +693.553, Z    +0.000, E1   +58.665, E3 -234812.979}
SPL {X  -157.294, Y  +700.745, Z    +0.000, E1   +58.469, E3 -234823.429}
SPL {X  -156.031, Y  +706.871, Z    +0.000, E1   +58.260, E3 -234832.575}
SPL {X  -154.558, Y  +712.835, Z    +0.000, E1   +58.028, E3 -234841.702}
SPL {X  -152.750, Y  +719.085, Z    +0.000, E1   +57.721, E3 -234851.548}
SPL {X  -150.741, Y  +725.111, Z    +0.000, E1   +57.387, E3 -234861.252}
SPL {X  -148.665, Y  +730.623, Z    +0.000, E1   +57.007, E3 -234870.401}
SPL {X  -146.664, Y  +735.425, Z    +0.000, E1   +56.657, E3 -234878.491}
SPL {X  -144.631, Y  +739.900, Z    +0.000, E1   +56.280, E3 -234886.176}
SPL {X  -141.795, Y  +745.600, Z    +0.000, E1   +55.801, E3 -234896.059}
SPL {X  -138.492, Y  +751.605, Z    +0.000, E1   +55.137, E3 -234906.783}
SPL {X  -124.324, Y  +772.199, Z    +0.000, E1   +48.708, E3 -234985.791}
ENDSPLINE

SPLINE
SPL {X  -129.118, Y  +765.975, Z    +0.000, E1   +43.713, E3 -235050.276}
SPL {X  -146.252, Y  +736.362, Z    +0.000, E1   +34.795, E3 -235099.454}
SPL {X  -155.916, Y  +707.374, Z    +0.000, E1   +22.878, E3 -235116.339}
SPL {X  -159.039, Y  +688.920, Z    +0.000, E1   +13.016, E3 -235121.574}
SPL {X  -159.888, Y  +677.224, Z    +0.000, E1    +5.773, E3 -235123.287}
SPL {X  -159.990, Y  +670.275, Z    +0.000, E1    +0.854, E3 -235123.740}
SPL {X  -159.990, Y  +667.097, Z    +0.000, E1    -2.190, E3 -235123.858}
SPL {X  -159.990, Y  +662.904, Z    +0.000, E1    -7.618, E3 -235124.146}
SPL {X  -159.990, Y  +658.509, Z    +0.000, E1   -13.882, E3 -235124.682}
SPL {X  -159.990, Y  +652.317, Z    +0.000, E1   -22.778, E3 -235125.817}
SPL {X  -159.990, Y  +640.689, Z    +0.000, E1   -37.390, E3 -235127.360}
SPL {X  -159.990, Y  +585.634, Z    +0.000, E1   -68.681, E3 -235127.984}
SPL {X  -159.990, Y  +457.771, Z    +0.000, E1   -68.079, E3 -235218.545}
SPL {X  -159.990, Y  +453.218, Z    +0.000, E1   -67.322, E3 -235228.981}
SPL {X  -159.990, Y  +450.256, Z    +0.000, E1   -66.188, E3 -235240.913}
SPL {X  -159.990, Y  +445.667, Z    +0.000, E1   -65.356, E3 -235251.825}
SPL {X  -159.990, Y  +439.738, Z    +0.000, E1   -64.716, E3 -235262.638}
SPL {X  -159.990, Y  +435.528, Z    +0.000, E1   -63.972, E3 -235272.514}
SPL {X  -159.990, Y  +429.021, Z    +0.000, E1   -63.228, E3 -235285.126}
SPL {X  -159.990, Y  +423.267, Z    +0.000, E1   -62.365, E3 -235297.424}
SPL {X  -159.990, Y  +418.218, Z    +0.000, E1   -61.769, E3 -235307.437}
SPL {X  -159.990, Y  +412.274, Z    +0.000, E1   -61.123, E3 -235318.841}
SPL {X  -159.990, Y  +408.631, Z    +0.000, E1   -60.233, E3 -235329.303}
SPL {X  -159.990, Y  +402.821, Z    +0.000, E1   -59.334, E3 -235342.831}
SPL {X  -159.990, Y  +395.849, Z    +0.000, E1   -58.799, E3 -235355.095}
SPL {X  -159.990, Y  +387.403, Z    +0.000, E1   -58.805, E3 -235365.941}
SPL {X  -159.948, Y  +378.844, Z    +0.000, E1   -58.798, E3 -235376.981}
SPL {X  -159.570, Y  +370.916, Z    +0.000, E1   -58.738, E3 -235387.576}
SPL {X  -158.865, Y  +363.563, Z    +0.000, E1   -58.615, E3 -235397.786}
SPL {X  -157.976, Y  +357.197, Z    +0.000, E1   -58.476, E3 -235406.886}
SPL {X  -156.730, Y  +350.368, Z    +0.000, E1   -58.276, E3 -235416.982}
SPL {X  -155.026, Y  +342.956, Z    +0.000, E1   -58.003, E3 -235428.254}
SPL {X  -152.946, Y  +335.551, Z    +0.000, E1   -57.653, E3 -235439.902}
SPL {X  -150.105, Y  +327.135, Z    +0.000, E1   -57.196, E3 -235453.522}
SPL {X  -146.578, Y  +318.377, Z    +0.000, E1   -56.572, E3 -235468.215}
SPL {X  -143.463, Y  +311.683, Z    +0.000, E1   -55.972, E3 -235479.828}
SPL {X  -140.858, Y  +306.633, Z    +0.000, E1   -55.477, E3 -235488.746}
SPL {X  -138.338, Y  +302.130, Z    +0.000, E1   -54.992, E3 -235496.795}
SPL {X  -124.427, Y  +281.929, Z    +0.000, E1   -46.852, E3 -235601.032}
ENDSPLINE

SPLINE
SPL {X  -148.251, Y  +322.346, Z    +0.000, E1   -33.039, E3 -235688.957}
SPL {X  -157.534, Y  +354.574, Z    +0.000, E1   -18.815, E3 -235705.786}
SPL {X  -159.548, Y  +370.614, Z    +0.000, E1    -9.656, E3 -235709.411}
SPL {X  -159.928, Y  +378.035, Z    +0.000, E1    -4.866, E3 -235710.327}
SPL {X  -159.990, Y  +383.381, Z    +0.000, E1    -1.123, E3 -235710.647}
SPL {X  -159.990, Y  +386.348, Z    +0.000, E1    +1.571, E3 -235710.756}
SPL {X  -159.990, Y  +391.422, Z    +0.000, E1    +7.757, E3 -235711.130}
SPL {X  -159.990, Y  +396.843, Z    +0.000, E1   +15.720, E3 -235711.792}
SPL {X  -159.990, Y  +403.976, Z    +0.000, E1   +25.456, E3 -235713.330}
SPL {X  -159.990, Y  +417.120, Z    +0.000, E1   +39.678, E3 -235717.361}
SPL {X  -159.990, Y  +456.927, Z    +0.000, E1   +55.382, E3 -235739.222}
SPL {X  -159.990, Y  +530.047, Z    +0.000, E1   +58.901, E3 -235809.056}
SPL {X  -159.990, Y  +538.035, Z    +0.000, E1   +58.900, E3 -235819.281}
SPL {X  -159.990, Y  +546.883, Z    +0.000, E1   +58.912, E3 -235830.585}
SPL {X  -159.990, Y  +555.949, Z    +0.000, E1   +58.900, E3 -235842.204}
SPL {X  -159.990, Y  +563.718, Z    +0.000, E1   +58.903, E3 -235852.124}
SPL {X  -159.990, Y  +571.529, Z    +0.000, E1   +58.906, E3 -235862.108}
SPL {X  -159.990, Y  +579.859, Z    +0.000, E1   +58.907, E3 -235872.768}
SPL {X  -159.990, Y  +588.526, Z    +0.000, E1   +58.910, E3 -235883.841}
SPL {X  -159.990, Y  +596.521, Z    +0.000, E1   +58.902, E3 -235894.100}
SPL {X  -159.990, Y  +605.444, Z    +0.000, E1   +58.918, E3 -235905.490}
SPL {X  -159.990, Y  +613.908, Z    +0.000, E1   +58.900, E3 -235916.349}
SPL {X  -159.990, Y  +621.342, Z    +0.000, E1   +58.904, E3 -235925.857}
SPL {X  -159.990, Y  +629.920, Z    +0.000, E1   +58.912, E3 -235936.830}
SPL {X  -159.990, Y  +642.398, Z    +0.000, E1   +58.947, E3 -235952.737}
SPL {X  -159.990, Y  +654.206, Z    +0.000, E1   +58.908, E3 -235967.908}
SPL {X  -159.990, Y  +661.562, Z    +0.000, E1   +58.900, E3 -235977.336}
SPL {X  -159.990, Y  +670.328, Z    +0.000, E1   +58.911, E3 -235988.536}
SPL {X  -159.795, Y  +679.404, Z    +0.000, E1   +58.876, E3 -236000.361}
SPL {X  -159.282, Y  +686.534, Z    +0.000, E1   +58.787, E3 -236010.035}
SPL {X  -158.463, Y  +693.553, Z    +0.000, E1   +58.665, E3 -236019.876}
SPL {X  -157.294, Y  +700.745, Z    +0.000, E1   +58.469, E3 -236030.326}
SPL {X  -156.031, Y  +706.871, Z    +0.000, E1   +58.260, E3 -236039.471}
SPL {X  -154.558, Y  +712.835, Z    +0.000, E1   +58.028, E3 -236048.599}
SPL {X  -152.750, Y  +719.085, Z    +0.000, E1   +57.721, E3 -236058.445}
SPL {X  -150.741, Y  +725.111, Z    +0.000, E1   +57.387, E3 -236068.149}
SPL {X  -148.665, Y  +730.623, Z    +0.000, E1   +57.007, E3 -236077.297}
SPL {X  -146.664, Y  +735.425, Z    +0.000, E1   +56.657, E3 -236085.388}
SPL {X  -144.631, Y  +739.900, Z    +0.000, E1   +56.280, E3 -236093.073}
SPL {X  -141.795, Y  +745.600, Z    +0.000, E1   +55.801, E3 -236102.956}
SPL {X  -138.492, Y  +751.605, Z    +0.000, E1   +55.137, E3 -236113.679}
SPL {X  -124.324, Y  +772.199, Z    +0.000, E1   +48.708, E3 -236192.687}
ENDSPLINE

SPLINE
SPL {X  -129.118, Y  +765.975, Z    +0.000, E1   +43.713, E3 -236257.173}
SPL {X  -146.252, Y  +736.362, Z    +0.000, E1   +34.795, E3 -236306.350}
SPL {X  -154.088, Y  +714.555, Z    +0.000, E1   +26.177, E3 -236320.367}
SPL {X  -156.688, Y  +703.837, Z    +0.000, E1   +21.096, E3 -236324.539}
SPL {X  -159.039, Y  +688.920, Z    +0.000, E1   +13.016, E3 -236328.470}
SPL {X  -159.888, Y  +677.224, Z    +0.000, E1    +5.773, E3 -236330.183}
SPL {X  -159.990, Y  +671.755, Z    +0.000, E1    +1.905, E3 -236330.587}
SPL {X  -159.990, Y  +669.598, Z    +0.000, E1    +0.205, E3 -236330.660}
SPL {X  -159.990, Y  +667.097, Z    +0.000, E1    -2.190, E3 -236330.755}
SPL {X  -159.990, Y  +662.904, Z    +0.000, E1    -7.618, E3 -236331.043}
SPL {X  -159.990, Y  +658.509, Z    +0.000, E1   -13.882, E3 -236331.579}
SPL {X  -159.990, Y  +652.317, Z    +0.000, E1   -22.778, E3 -236332.714}
SPL {X  -159.990, Y  +640.689, Z    +0.000, E1   -37.390, E3 -236334.257}
SPL {X  -159.990, Y  +585.634, Z    +0.000, E1   -68.681, E3 -236334.881}
SPL {X  -159.990, Y  +457.771, Z    +0.000, E1   -68.079, E3 -236425.442}
SPL {X  -159.990, Y  +453.218, Z    +0.000, E1   -67.322, E3 -236435.877}
SPL {X  -159.990, Y  +450.256, Z    +0.000, E1   -66.188, E3 -236447.810}
SPL {X  -159.990, Y  +445.667, Z    +0.000, E1   -65.356, E3 -236458.722}
SPL {X  -159.990, Y  +439.738, Z    +0.000, E1   -64.716, E3 -236469.535}
SPL {X  -159.990, Y  +435.528, Z    +0.000, E1   -63.972, E3 -236479.410}
SPL {X  -159.990, Y  +429.021, Z    +0.000, E1   -63.228, E3 -236492.023}
SPL {X  -159.990, Y  +423.267, Z    +0.000, E1   -62.365, E3 -236504.321}
SPL {X  -159.990, Y  +418.218, Z    +0.000, E1   -61.769, E3 -236514.334}
SPL {X  -159.990, Y  +412.274, Z    +0.000, E1   -61.123, E3 -236525.737}
SPL {X  -159.990, Y  +408.631, Z    +0.000, E1   -60.233, E3 -236536.200}
SPL {X  -159.990, Y  +404.834, Z    +0.000, E1   -59.529, E3 -236545.655}
SPL {X  -159.990, Y  +397.866, Z    +0.000, E1   -58.924, E3 -236558.742}
SPL {X  -159.990, Y  +387.403, Z    +0.000, E1   -58.805, E3 -236572.838}
SPL {X  -159.948, Y  +378.844, Z    +0.000, E1   -58.798, E3 -236583.877}
SPL {X  -159.570, Y  +370.916, Z    +0.000, E1   -58.738, E3 -236594.473}
SPL {X  -158.865, Y  +363.563, Z    +0.000, E1   -58.615, E3 -236604.682}
SPL {X  -157.976, Y  +357.197, Z    +0.000, E1   -58.476, E3 -236613.783}
SPL {X  -156.730, Y  +350.368, Z    +0.000, E1   -58.276, E3 -236623.878}
SPL {X  -155.026, Y  +342.956, Z    +0.000, E1   -58.003, E3 -236635.150}
SPL {X  -152.946, Y  +335.551, Z    +0.000, E1   -57.653, E3 -236646.798}
SPL {X  -150.899, Y  +329.336, Z    +0.000, E1   -57.290, E3 -236656.864}
SPL {X  -149.179, Y  +324.687, Z    +0.000, E1   -56.983, E3 -236664.553}
SPL {X  -147.281, Y  +320.009, Z    +0.000, E1   -56.662, E3 -236672.379}
SPL {X  -144.114, Y  +313.017, Z    +0.000, E1   -56.131, E3 -236684.347}
SPL {X  -140.858, Y  +306.633, Z    +0.000, E1   -55.477, E3 -236695.642}
SPL {X  -138.338, Y  +302.130, Z    +0.000, E1   -54.992, E3 -236703.692}
SPL {X  -124.427, Y  +281.929, Z    +0.000, E1   -46.852, E3 -236807.928}
ENDSPLINE

SPLINE
SPL {X  -148.251, Y  +322.346, Z    +0.000, E1   -33.039, E3 -236895.853}
SPL {X  -157.534, Y  +354.574, Z    +0.000, E1   -18.815, E3 -236912.682}
SPL {X  -159.548, Y  +370.614, Z    +0.000, E1    -9.656, E3 -236916.308}
SPL {X  -159.973, Y  +380.173, Z    +0.000, E1    -3.469, E3 -236917.375}
SPL {X  -159.990, Y  +384.791, Z    +0.000, E1    +0.055, E3 -236917.594}
SPL {X  -159.990, Y  +388.179, Z    +0.000, E1    +3.660, E3 -236917.754}
SPL {X  -159.990, Y  +394.222, Z    +0.000, E1   +11.674, E3 -236918.347}
SPL {X  -159.990, Y  +403.976, Z    +0.000, E1   +25.456, E3 -236920.227}
SPL {X  -159.990, Y  +417.120, Z    +0.000, E1   +39.678, E3 -236924.258}
SPL {X  -159.990, Y  +456.927, Z    +0.000, E1   +55.382, E3 -236946.118}
SPL {X  -159.990, Y  +530.047, Z    +0.000, E1   +58.901, E3 -237015.952}
SPL {X  -159.990, Y  +538.035, Z    +0.000, E1   +58.900, E3 -237026.178}
SPL {X  -159.990, Y  +546.883, Z    +0.000, E1   +58.912, E3 -237037.481}
SPL {X  -159.990, Y  +555.949, Z    +0.000, E1   +58.900, E3 -237049.101}
SPL {X  -159.990, Y  +563.718, Z    +0.000, E1   +58.903, E3 -237059.021}
SPL {X  -159.990, Y  +571.529, Z    +0.000, E1   +58.906, E3 -237069.005}
SPL {X  -159.990, Y  +579.859, Z    +0.000, E1   +58.907, E3 -237079.664}
SPL {X  -159.990, Y  +588.526, Z    +0.000, E1   +58.910, E3 -237090.738}
SPL {X  -159.990, Y  +596.521, Z    +0.000, E1   +58.902, E3 -237100.997}
SPL {X  -159.990, Y  +605.444, Z    +0.000, E1   +58.918, E3 -237112.386}
SPL {X  -159.990, Y  +613.908, Z    +0.000, E1   +58.900, E3 -237123.246}
SPL {X  -159.990, Y  +621.342, Z    +0.000, E1   +58.904, E3 -237132.754}
SPL {X  -159.990, Y  +629.920, Z    +0.000, E1   +58.912, E3 -237143.726}
SPL {X  -159.990, Y  +642.398, Z    +0.000, E1   +58.947, E3 -237159.634}
SPL {X  -159.990, Y  +654.206, Z    +0.000, E1   +58.908, E3 -237174.805}
SPL {X  -159.990, Y  +661.562, Z    +0.000, E1   +58.900, E3 -237184.233}
SPL {X  -159.990, Y  +670.328, Z    +0.000, E1   +58.911, E3 -237195.432}
SPL {X  -159.795, Y  +679.404, Z    +0.000, E1   +58.876, E3 -237207.257}
SPL {X  -159.282, Y  +686.534, Z    +0.000, E1   +58.787, E3 -237216.931}
SPL {X  -158.463, Y  +693.553, Z    +0.000, E1   +58.665, E3 -237226.772}
SPL {X  -157.294, Y  +700.745, Z    +0.000, E1   +58.469, E3 -237237.222}
SPL {X  -156.031, Y  +706.871, Z    +0.000, E1   +58.260, E3 -237246.368}
SPL {X  -154.558, Y  +712.835, Z    +0.000, E1   +58.028, E3 -237255.495}
SPL {X  -152.750, Y  +719.085, Z    +0.000, E1   +57.721, E3 -237265.341}
SPL {X  -150.741, Y  +725.111, Z    +0.000, E1   +57.387, E3 -237275.045}
SPL {X  -148.665, Y  +730.623, Z    +0.000, E1   +57.007, E3 -237284.194}
SPL {X  -146.664, Y  +735.425, Z    +0.000, E1   +56.657, E3 -237292.284}
SPL {X  -143.496, Y  +742.251, Z    +0.000, E1   +56.124, E3 -237303.977}
SPL {X  -140.752, Y  +747.564, Z    +0.000, E1   +55.554, E3 -237313.385}
SPL {X  -138.492, Y  +751.605, Z    +0.000, E1   +55.137, E3 -237320.576}
SPL {X  -124.324, Y  +772.199, Z    +0.000, E1   +48.708, E3 -237399.584}
ENDSPLINE

SPLINE
SPL {X  -129.118, Y  +765.975, Z    +0.000, E1   +43.713, E3 -237464.069}
SPL {X  -146.252, Y  +736.362, Z    +0.000, E1   +34.795, E3 -237513.247}
SPL {X  -155.916, Y  +707.374, Z    +0.000, E1   +22.878, E3 -237530.133}
SPL {X  -159.039, Y  +688.920, Z    +0.000, E1   +13.016, E3 -237535.367}
SPL {X  -159.777, Y  +679.762, Z    +0.000, E1    +7.372, E3 -237536.822}
SPL {X  -159.984, Y  +672.872, Z    +0.000, E1    +2.784, E3 -237537.419}
SPL {X  -159.990, Y  +668.898, Z    +0.000, E1    -0.346, E3 -237537.577}
SPL {X  -159.990, Y  +666.084, Z    +0.000, E1    -3.512, E3 -237537.700}
SPL {X  -159.990, Y  +662.904, Z    +0.000, E1    -7.618, E3 -237537.939}
SPL {X  -159.990, Y  +658.509, Z    +0.000, E1   -13.882, E3 -237538.475}
SPL {X  -159.990, Y  +652.317, Z    +0.000, E1   -22.778, E3 -237539.610}
SPL {X  -159.990, Y  +640.689, Z    +0.000, E1   -37.390, E3 -237541.153}
SPL {X  -159.990, Y  +585.634, Z    +0.000, E1   -68.681, E3 -237541.777}
SPL {X  -159.990, Y  +457.771, Z    +0.000, E1   -68.079, E3 -237632.339}
SPL {X  -159.990, Y  +453.218, Z    +0.000, E1   -67.322, E3 -237642.774}
SPL {X  -159.990, Y  +450.256, Z    +0.000, E1   -66.188, E3 -237654.707}
SPL {X  -159.990, Y  +445.667, Z    +0.000, E1   -65.356, E3 -237665.618}
SPL {X  -159.990, Y  +439.738, Z    +0.000, E1   -64.716, E3 -237676.431}
SPL {X  -159.990, Y  +433.217, Z    +0.000, E1   -63.756, E3 -237690.575}
SPL {X  -159.990, Y  +425.111, Z    +0.000, E1   -62.687, E3 -237707.116}
SPL {X  -159.990, Y  +418.218, Z    +0.000, E1   -61.769, E3 -237721.230}
SPL {X  -159.990, Y  +412.274, Z    +0.000, E1   -61.123, E3 -237732.634}
SPL {X  -159.990, Y  +408.631, Z    +0.000, E1   -60.233, E3 -237743.096}
SPL {X  -159.990, Y  +402.821, Z    +0.000, E1   -59.334, E3 -237756.624}
SPL {X  -159.990, Y  +395.849, Z    +0.000, E1   -58.799, E3 -237768.888}
SPL {X  -159.990, Y  +387.403, Z    +0.000, E1   -58.805, E3 -237779.734}
SPL {X  -159.948, Y  +378.844, Z    +0.000, E1   -58.798, E3 -237790.774}
SPL {X  -159.570, Y  +370.916, Z    +0.000, E1   -58.738, E3 -237801.369}
SPL {X  -158.865, Y  +363.563, Z    +0.000, E1   -58.615, E3 -237811.579}
SPL {X  -157.976, Y  +357.197, Z    +0.000, E1   -58.476, E3 -237820.679}
SPL {X  -156.730, Y  +350.368, Z    +0.000, E1   -58.276, E3 -237830.775}
SPL {X  -155.026, Y  +342.956, Z    +0.000, E1   -58.003, E3 -237842.047}
SPL {X  -152.946, Y  +335.551, Z    +0.000, E1   -57.653, E3 -237853.695}
SPL {X  -150.105, Y  +327.135, Z    +0.000, E1   -57.196, E3 -237867.315}
SPL {X  -146.578, Y  +318.377, Z    +0.000, E1   -56.572, E3 -237882.008}
SPL {X  -143.463, Y  +311.683, Z    +0.000, E1   -55.972, E3 -237893.621}
SPL {X  -140.858, Y  +306.633, Z    +0.000, E1   -55.477, E3 -237902.539}
SPL {X  -138.338, Y  +302.130, Z    +0.000, E1   -54.992, E3 -237910.588}
SPL {X  -124.427, Y  +281.929, Z    +0.000, E1   -46.852, E3 -238014.825}
ENDSPLINE

SPLINE
SPL {X  -148.251, Y  +322.346, Z    +0.000, E1   -33.039, E3 -238102.750}
SPL {X  -157.534, Y  +354.574, Z    +0.000, E1   -18.815, E3 -238119.579}
SPL {X  -159.548, Y  +370.614, Z    +0.000, E1    -9.656, E3 -238123.204}
SPL {X  -159.973, Y  +380.173, Z    +0.000, E1    -3.469, E3 -238124.271}
SPL {X  -159.990, Y  +384.078, Z    +0.000, E1    -0.490, E3 -238124.469}
SPL {X  -159.990, Y  +385.440, Z    +0.000, E1    +0.747, E3 -238124.509}
SPL {X  -159.990, Y  +388.179, Z    +0.000, E1    +3.660, E3 -238124.650}
SPL {X  -159.990, Y  +394.222, Z    +0.000, E1   +11.674, E3 -238125.244}
SPL {X  -159.990, Y  +403.976, Z    +0.000, E1   +25.456, E3 -238127.123}
SPL {X  -159.990, Y  +417.120, Z    +0.000, E1   +39.678, E3 -238131.155}
SPL {X  -159.990, Y  +456.927, Z    +0.000, E1   +55.382, E3 -238153.015}
SPL {X  -159.990, Y  +530.047, Z    +0.000, E1   +58.901, E3 -238222.849}
SPL {X  -159.990, Y  +538.035, Z    +0.000, E1   +58.900, E3 -238233.074}
SPL {X  -159.990, Y  +546.883, Z    +0.000, E1   +58.912, E3 -238244.378}
SPL {X  -159.990, Y  +555.949, Z    +0.000, E1   +58.900, E3 -238255.997}
SPL {X  -159.990, Y  +563.718, Z    +0.000, E1   +58.903, E3 -238265.917}
SPL {X  -159.990, Y  +571.529, Z    +0.000, E1   +58.906, E3 -238275.901}
SPL {X  -159.990, Y  +579.859, Z    +0.000, E1   +58.907, E3 -238286.561}
SPL {X  -159.990, Y  +588.526, Z    +0.000, E1   +58.910, E3 -238297.634}
SPL {X  -159.990, Y  +596.521, Z    +0.000, E1   +58.902, E3 -238307.893}
SPL {X  -159.990, Y  +605.444, Z    +0.000, E1   +58.918, E3 -238319.283}
SPL {X  -159.990, Y  +618.101, Z    +0.000, E1   +58.946, E3 -238335.430}
SPL {X  -159.990, Y  +629.920, Z    +0.000, E1   +58.912, E3 -238350.623}
SPL {X  -159.990, Y  +638.424, Z    +0.000, E1   +58.901, E3 -238361.523}
SPL {X  -159.990, Y  +645.995, Z    +0.000, E1   +58.900, E3 -238371.211}
SPL {X  -159.990, Y  +654.206, Z    +0.000, E1   +58.908, E3 -238381.701}
SPL {X  -159.990, Y  +661.562, Z    +0.000, E1   +58.900, E3 -238391.130}
SPL {X  -159.990, Y  +670.328, Z    +0.000, E1   +58.911, E3 -238402.329}
SPL {X  -159.795, Y  +679.404, Z    +0.000, E1   +58.876, E3 -238414.154}
SPL {X  -159.282, Y  +686.534, Z    +0.000, E1   +58.787, E3 -238423.828}
SPL {X  -158.463, Y  +693.553, Z    +0.000, E1   +58.665, E3 -238433.669}
SPL {X  -157.294, Y  +700.745, Z    +0.000, E1   +58.469, E3 -238444.119}
SPL {X  -156.031, Y  +706.871, Z    +0.000, E1   +58.260, E3 -238453.265}
SPL {X  -154.558, Y  +712.835, Z    +0.000, E1   +58.028, E3 -238462.392}
SPL {X  -152.750, Y  +719.085, Z    +0.000, E1   +57.721, E3 -238472.238}
SPL {X  -150.741, Y  +725.111, Z    +0.000, E1   +57.387, E3 -238481.942}
SPL {X  -148.665, Y  +730.623, Z    +0.000, E1   +57.007, E3 -238491.091}
SPL {X  -146.664, Y  +735.425, Z    +0.000, E1   +56.657, E3 -238499.181}
SPL {X  -143.496, Y  +742.251, Z    +0.000, E1   +56.124, E3 -238510.874}
SPL {X  -140.752, Y  +747.564, Z    +0.000, E1   +55.554, E3 -238520.281}
SPL {X  -138.492, Y  +751.605, Z    +0.000, E1   +55.137, E3 -238527.472}
SPL {X  -124.324, Y  +772.199, Z    +0.000, E1   +48.708, E3 -238606.480}
ENDSPLINE

SPLINE
SPL {X  -129.118, Y  +765.975, Z    +0.000, E1   +43.713, E3 -238670.966}
SPL {X  -146.252, Y  +736.362, Z    +0.000, E1   +34.795, E3 -238720.144}
SPL {X  -155.916, Y  +707.374, Z    +0.000, E1   +22.878, E3 -238737.029}
SPL {X  -159.039, Y  +688.920, Z    +0.000, E1   +13.016, E3 -238742.264}
SPL {X  -159.888, Y  +677.224, Z    +0.000, E1    +5.773, E3 -238743.976}
SPL {X  -159.990, Y  +671.755, Z    +0.000, E1    +1.905, E3 -238744.380}
SPL {X  -159.990, Y  +669.598, Z    +0.000, E1    +0.205, E3 -238744.453}
SPL {X  -159.990, Y  +667.097, Z    +0.000, E1    -2.190, E3 -238744.548}
SPL {X  -159.990, Y  +662.904, Z    +0.000, E1    -7.618, E3 -238744.836}
SPL {X  -159.990, Y  +658.509, Z    +0.000, E1   -13.882, E3 -238745.372}
SPL {X  -159.990, Y  +652.317, Z    +0.000, E1   -22.778, E3 -238746.507}
SPL {X  -159.990, Y  +640.689, Z    +0.000, E1   -37.390, E3 -238748.050}
SPL {X  -159.990, Y  +585.634, Z    +0.000, E1   -68.681, E3 -238748.674}
SPL {X  -159.990, Y  +457.771, Z    +0.000, E1   -68.079, E3 -238839.235}
SPL {X  -159.990, Y  +453.218, Z    +0.000, E1   -67.322, E3 -238849.670}
SPL {X  -159.990, Y  +450.256, Z    +0.000, E1   -66.188, E3 -238861.603}
SPL {X  -159.990, Y  +445.667, Z    +0.000, E1   -65.356, E3 -238872.515}
SPL {X  -159.990, Y  +439.738, Z    +0.000, E1   -64.716, E3 -238883.328}
SPL {X  -159.990, Y  +435.528, Z    +0.000, E1   -63.972, E3 -238893.203}
SPL {X  -159.990, Y  +429.021, Z    +0.000, E1   -63.228, E3 -238905.816}
SPL {X  -159.990, Y  +423.267, Z    +0.000, E1   -62.365, E3 -238918.114}
SPL {X  -159.990, Y  +418.218, Z    +0.000, E1   -61.769, E3 -238928.127}
SPL {X  -159.990, Y  +412.274, Z    +0.000, E1   -61.123, E3 -238939.531}
SPL {X  -159.990, Y  +408.631, Z    +0.000, E1   -60.233, E3 -238949.993}
SPL {X  -159.990, Y  +404.834, Z    +0.000, E1   -59.529, E3 -238959.448}
SPL {X  -159.990, Y  +397.866, Z    +0.000, E1   -58.924, E3 -238972.535}
SPL {X  -159.990, Y  +387.403, Z    +0.000, E1   -58.805, E3 -238986.631}
SPL {X  -159.948, Y  +378.844, Z    +0.000, E1   -58.798, E3 -238997.670}
SPL {X  -159.570, Y  +370.916, Z    +0.000, E1   -58.738, E3 -239008.266}
SPL {X  -158.865, Y  +363.563, Z    +0.000, E1   -58.615, E3 -239018.475}
SPL {X  -157.976, Y  +357.197, Z    +0.000, E1   -58.476, E3 -239027.576}
SPL {X  -156.730, Y  +350.368, Z    +0.000, E1   -58.276, E3 -239037.671}
SPL {X  -155.026, Y  +342.956, Z    +0.000, E1   -58.003, E3 -239048.943}
SPL {X  -152.946, Y  +335.551, Z    +0.000, E1   -57.653, E3 -239060.591}
SPL {X  -150.105, Y  +327.135, Z    +0.000, E1   -57.196, E3 -239074.212}
SPL {X  -146.578, Y  +318.377, Z    +0.000, E1   -56.572, E3 -239088.904}
SPL {X  -143.463, Y  +311.683, Z    +0.000, E1   -55.972, E3 -239100.518}
SPL {X  -140.858, Y  +306.633, Z    +0.000, E1   -55.477, E3 -239109.435}
SPL {X  -138.338, Y  +302.130, Z    +0.000, E1   -54.992, E3 -239117.485}
SPL {X  -124.427, Y  +281.929, Z    +0.000, E1   -46.852, E3 -239221.721}
ENDSPLINE

SPLINE
SPL {X  -148.251, Y  +322.346, Z    +0.000, E1   -33.039, E3 -239309.646}
SPL {X  -157.534, Y  +354.574, Z    +0.000, E1   -18.815, E3 -239326.475}
SPL {X  -159.548, Y  +370.614, Z    +0.000, E1    -9.656, E3 -239330.101}
SPL {X  -159.928, Y  +378.035, Z    +0.000, E1    -4.866, E3 -239331.016}
SPL {X  -159.990, Y  +383.381, Z    +0.000, E1    -1.123, E3 -239331.337}
SPL {X  -159.990, Y  +386.348, Z    +0.000, E1    +1.571, E3 -239331.446}
SPL {X  -159.990, Y  +391.422, Z    +0.000, E1    +7.757, E3 -239331.820}
SPL {X  -159.990, Y  +399.099, Z    +0.000, E1   +18.787, E3 -239332.927}
SPL {X  -159.990, Y  +406.316, Z    +0.000, E1   +28.569, E3 -239334.604}
SPL {X  -159.990, Y  +417.120, Z    +0.000, E1   +39.678, E3 -239338.051}
SPL {X  -159.990, Y  +456.927, Z    +0.000, E1   +55.382, E3 -239359.911}
SPL {X  -159.990, Y  +530.047, Z    +0.000, E1   +58.901, E3 -239429.745}
SPL {X  -159.990, Y  +538.035, Z    +0.000, E1   +58.900, E3 -239439.971}
SPL {X  -159.990, Y  +546.883, Z    +0.000, E1   +58.912, E3 -239451.274}
SPL {X  -159.990, Y  +555.949, Z    +0.000, E1   +58.900, E3 -239462.894}
SPL {X  -159.990, Y  +563.718, Z    +0.000, E1   +58.903, E3 -239472.814}
SPL {X  -159.990, Y  +571.529, Z    +0.000, E1   +58.906, E3 -239482.798}
SPL {X  -159.990, Y  +579.859, Z    +0.000, E1   +58.907, E3 -239493.457}
SPL {X  -159.990, Y  +588.526, Z    +0.000, E1   +58.910, E3 -239504.531}
SPL {X  -159.990, Y  +596.521, Z    +0.000, E1   +58.902, E3 -239514.790}
SPL {X  -159.990, Y  +605.444, Z    +0.000, E1   +58.918, E3 -239526.179}
SPL {X  -159.990, Y  +618.101, Z    +0.000, E1   +58.946, E3 -239542.326}
SPL {X  -159.990, Y  +629.920, Z    +0.000, E1   +58.912, E3 -239557.519}
SPL {X  -159.990, Y  +638.424, Z    +0.000, E1   +58.901, E3 -239568.419}
SPL {X  -159.990, Y  +645.995, Z    +0.000, E1   +58.900, E3 -239578.107}
SPL {X  -159.990, Y  +654.206, Z    +0.000, E1   +58.908, E3 -239588.598}
SPL {X  -159.990, Y  +661.562, Z    +0.000, E1   +58.900, E3 -239598.026}
SPL {X  -159.990, Y  +670.328, Z    +0.000, E1   +58.911, E3 -239609.225}
SPL {X  -159.795, Y  +679.404, Z    +0.000, E1   +58.876, E3 -239621.051}
SPL {X  -159.282, Y  +686.534, Z    +0.000, E1   +58.787, E3 -239630.724}
SPL {X  -158.463, Y  +693.553, Z    +0.000, E1   +58.665, E3 -239640.565}
SPL {X  -157.294, Y  +700.745, Z    +0.000, E1   +58.469, E3 -239651.015}
SPL {X  -156.031, Y  +706.871, Z    +0.000, E1   +58.260, E3 -239660.161}
SPL {X  -154.558, Y  +712.835, Z    +0.000, E1   +58.028, E3 -239669.288}
SPL {X  -152.750, Y  +719.085, Z    +0.000, E1   +57.721, E3 -239679.134}
SPL {X  -150.741, Y  +725.111, Z    +0.000, E1   +57.387, E3 -239688.838}
SPL {X  -148.665, Y  +730.623, Z    +0.000, E1   +57.007, E3 -239697.987}
SPL {X  -146.664, Y  +735.425, Z    +0.000, E1   +56.657, E3 -239706.077}
SPL {X  -143.496, Y  +742.251, Z    +0.000, E1   +56.124, E3 -239717.770}
SPL {X  -140.752, Y  +747.564, Z    +0.000, E1   +55.554, E3 -239727.178}
SPL {X  -138.492, Y  +751.605, Z    +0.000, E1   +55.137, E3 -239734.369}
SPL {X  -124.324, Y  +772.199, Z    +0.000, E1   +48.708, E3 -239813.377}
ENDSPLINE

SPLINE
SPL {X  -129.118, Y  +765.975, Z    +0.000, E1   +43.713, E3 -239877.862}
SPL {X  -146.252, Y  +736.362, Z    +0.000, E1   +34.795, E3 -239927.040}
SPL {X  -154.088, Y  +714.555, Z    +0.000, E1   +26.177, E3 -239941.056}
SPL {X  -156.688, Y  +703.837, Z    +0.000, E1   +21.096, E3 -239945.228}
SPL {X  -159.039, Y  +688.920, Z    +0.000, E1   +13.016, E3 -239949.160}
SPL {X  -159.888, Y  +677.224, Z    +0.000, E1    +5.773, E3 -239950.873}
SPL {X  -159.990, Y  +670.275, Z    +0.000, E1    +0.854, E3 -239951.327}
SPL {X  -159.990, Y  +667.097, Z    +0.000, E1    -2.190, E3 -239951.444}
SPL {X  -159.990, Y  +662.904, Z    +0.000, E1    -7.618, E3 -239951.732}
SPL {X  -159.990, Y  +658.509, Z    +0.000, E1   -13.882, E3 -239952.268}
SPL {X  -159.990, Y  +652.317, Z    +0.000, E1   -22.778, E3 -239953.404}
SPL {X  -159.990, Y  +640.689, Z    +0.000, E1   -37.390, E3 -239954.946}
SPL {X  -159.990, Y  +585.634, Z    +0.000, E1   -68.681, E3 -239955.570}
SPL {X  -159.990, Y  +457.771, Z    +0.000, E1   -68.079, E3 -240046.132}
SPL {X  -159.990, Y  +453.218, Z    +0.000, E1   -67.322, E3 -240056.567}
SPL {X  -159.990, Y  +450.256, Z    +0.000, E1   -66.188, E3 -240068.500}
SPL {X  -159.990, Y  +445.667, Z    +0.000, E1   -65.356, E3 -240079.411}
SPL {X  -159.990, Y  +439.738, Z    +0.000, E1   -64.716, E3 -240090.224}
SPL {X  -159.990, Y  +433.217, Z    +0.000, E1   -63.756, E3 -240104.369}
SPL {X  -159.990, Y  +425.111, Z    +0.000, E1   -62.687, E3 -240120.909}
SPL {X  -159.990, Y  +418.218, Z    +0.000, E1   -61.769, E3 -240135.023}
SPL {X  -159.990, Y  +412.274, Z    +0.000, E1   -61.123, E3 -240146.427}
SPL {X  -159.990, Y  +408.631, Z    +0.000, E1   -60.233, E3 -240156.890}
SPL {X  -159.990, Y  +404.834, Z    +0.000, E1   -59.529, E3 -240166.345}
SPL {X  -159.990, Y  +397.866, Z    +0.000, E1   -58.924, E3 -240179.432}
SPL {X  -159.990, Y  +387.403, Z    +0.000, E1   -58.805, E3 -240193.527}
SPL {X  -159.948, Y  +378.844, Z    +0.000, E1   -58.798, E3 -240204.567}
SPL {X  -159.570, Y  +370.916, Z    +0.000, E1   -58.738, E3 -240215.162}
SPL {X  -158.865, Y  +363.563, Z    +0.000, E1   -58.615, E3 -240225.372}
SPL {X  -157.976, Y  +357.197, Z    +0.000, E1   -58.476, E3 -240234.473}
SPL {X  -156.730, Y  +350.368, Z    +0.000, E1   -58.276, E3 -240244.568}
SPL {X  -155.026, Y  +342.956, Z    +0.000, E1   -58.003, E3 -240255.840}
SPL {X  -152.946, Y  +335.551, Z    +0.000, E1   -57.653, E3 -240267.488}
SPL {X  -150.105, Y  +327.135, Z    +0.000, E1   -57.196, E3 -240281.108}
SPL {X  -146.578, Y  +318.377, Z    +0.000, E1   -56.572, E3 -240295.801}
SPL {X  -143.463, Y  +311.683, Z    +0.000, E1   -55.972, E3 -240307.415}
SPL {X  -140.858, Y  +306.633, Z    +0.000, E1   -55.477, E3 -240316.332}
SPL {X  -138.338, Y  +302.130, Z    +0.000, E1   -54.992, E3 -240324.381}
SPL {X  -124.427, Y  +281.929, Z    +0.000, E1   -46.852, E3 -240428.618}
ENDSPLINE

SPLINE
SPL {X  -138.506, Y  +302.419, Z    +0.000, E1   -39.451, E3 -240494.592}
SPL {X  -149.686, Y  +326.013, Z    +0.000, E1   -31.658, E3 -240519.729}
SPL {X  -157.534, Y  +354.574, Z    +0.000, E1   -18.815, E3 -240533.372}
SPL {X  -159.548, Y  +370.614, Z    +0.000, E1    -9.656, E3 -240536.997}
SPL {X  -159.928, Y  +378.035, Z    +0.000, E1    -4.866, E3 -240537.913}
SPL {X  -159.988, Y  +381.742, Z    +0.000, E1    -2.273, E3 -240538.166}
SPL {X  -159.990, Y  +384.791, Z    +0.000, E1    +0.055, E3 -240538.283}
SPL {X  -159.990, Y  +388.179, Z    +0.000, E1    +3.660, E3 -240538.443}
SPL {X  -159.990, Y  +394.222, Z    +0.000, E1   +11.674, E3 -240539.037}
SPL {X  -159.990, Y  +403.976, Z    +0.000, E1   +25.456, E3 -240540.916}
SPL {X  -159.990, Y  +417.120, Z    +0.000, E1   +39.678, E3 -240544.948}
SPL {X  -159.990, Y  +456.927, Z    +0.000, E1   +55.382, E3 -240566.808}
SPL {X  -159.990, Y  +530.047, Z    +0.000, E1   +58.901, E3 -240636.642}
SPL {X  -159.990, Y  +538.035, Z    +0.000, E1   +58.900, E3 -240646.867}
SPL {X  -159.990, Y  +546.883, Z    +0.000, E1   +58.912, E3 -240658.171}
SPL {X  -159.990, Y  +555.949, Z    +0.000, E1   +58.900, E3 -240669.790}
SPL {X  -159.990, Y  +563.718, Z    +0.000, E1   +58.903, E3 -240679.710}
SPL {X  -159.990, Y  +571.529, Z    +0.000, E1   +58.906, E3 -240689.695}
SPL {X  -159.990, Y  +579.859, Z    +0.000, E1   +58.907, E3 -240700.354}
SPL {X  -159.990, Y  +588.526, Z    +0.000, E1   +58.910, E3 -240711.427}
SPL {X  -159.990, Y  +596.521, Z    +0.000, E1   +58.902, E3 -240721.687}
SPL {X  -159.990, Y  +605.444, Z    +0.000, E1   +58.918, E3 -240733.076}
SPL {X  -159.990, Y  +613.908, Z    +0.000, E1   +58.900, E3 -240743.935}
SPL {X  -159.990, Y  +621.342, Z    +0.000, E1   +58.904, E3 -240753.443}
SPL {X  -159.990, Y  +629.920, Z    +0.000, E1   +58.912, E3 -240764.416}
SPL {X  -159.990, Y  +642.398, Z    +0.000, E1   +58.947, E3 -240780.323}
SPL {X  -159.990, Y  +654.206, Z    +0.000, E1   +58.908, E3 -240795.494}
SPL {X  -159.990, Y  +661.562, Z    +0.000, E1   +58.900, E3 -240804.923}
SPL {X  -159.990, Y  +670.328, Z    +0.000, E1   +58.911, E3 -240816.122}
SPL {X  -159.795, Y  +679.404, Z    +0.000, E1   +58.876, E3 -240827.947}
SPL {X  -159.282, Y  +686.534, Z    +0.000, E1   +58.787, E3 -240837.621}
SPL {X  -158.463, Y  +693.553, Z    +0.000, E1   +58.665, E3 -240847.462}
SPL {X  -157.294, Y  +700.745, Z    +0.000, E1   +58.469, E3 -240857.912}
SPL {X  -156.031, Y  +706.871, Z    +0.000, E1   +58.260, E3 -240867.058}
SPL {X  -154.558, Y  +712.835, Z    +0.000, E1   +58.028, E3 -240876.185}
SPL {X  -152.750, Y  +719.085, Z    +0.000, E1   +57.721, E3 -240886.031}
SPL {X  -150.741, Y  +725.111, Z    +0.000, E1   +57.387, E3 -240895.735}
SPL {X  -148.665, Y  +730.623, Z    +0.000, E1   +57.007, E3 -240904.884}
SPL {X  -146.664, Y  +735.425, Z    +0.000, E1   +56.657, E3 -240912.974}
SPL {X  -144.631, Y  +739.900, Z    +0.000, E1   +56.280, E3 -240920.659}
SPL {X  -141.795, Y  +745.600, Z    +0.000, E1   +55.801, E3 -240930.542}
SPL {X  -138.492, Y  +751.605, Z    +0.000, E1   +55.137, E3 -240941.265}
SPL {X  -124.324, Y  +772.199, Z    +0.000, E1   +48.708, E3 -241020.274}
ENDSPLINE

SPLINE
SPL {X  -129.118, Y  +765.975, Z    +0.000, E1   +43.713, E3 -241084.759}
SPL {X  -146.252, Y  +736.362, Z    +0.000, E1   +34.795, E3 -241133.937}
SPL {X  -154.088, Y  +714.555, Z    +0.000, E1   +26.177, E3 -241147.953}
SPL {X  -156.688, Y  +703.837, Z    +0.000, E1   +21.096, E3 -241152.125}
SPL {X  -159.039, Y  +688.920, Z    +0.000, E1   +13.016, E3 -241156.057}
SPL {X  -159.888, Y  +677.224, Z    +0.000, E1    +5.773, E3 -241157.770}
SPL {X  -159.990, Y  +670.275, Z    +0.000, E1    +0.854, E3 -241158.223}
SPL {X  -159.990, Y  +667.097, Z    +0.000, E1    -2.190, E3 -241158.341}
SPL {X  -159.990, Y  +662.904, Z    +0.000, E1    -7.618, E3 -241158.629}
SPL {X  -159.990, Y  +658.509, Z    +0.000, E1   -13.882, E3 -241159.165}
SPL {X  -159.990, Y  +652.317, Z    +0.000, E1   -22.778, E3 -241160.300}
SPL {X  -159.990, Y  +640.689, Z    +0.000, E1   -37.390, E3 -241161.843}
SPL {X  -159.990, Y  +585.634, Z    +0.000, E1   -68.681, E3 -241162.467}
SPL {X  -159.990, Y  +457.771, Z    +0.000, E1   -68.079, E3 -241253.028}
SPL {X  -159.990, Y  +453.218, Z    +0.000, E1   -67.322, E3 -241263.463}
SPL {X  -159.990, Y  +450.256, Z    +0.000, E1   -66.188, E3 -241275.396}
SPL {X  -159.990, Y  +445.667, Z    +0.000, E1   -65.356, E3 -241286.308}
SPL {X  -159.990, Y  +439.738, Z    +0.000, E1   -64.716, E3 -241297.121}
SPL {X  -159.990, Y  +435.528, Z    +0.000, E1   -63.972, E3 -241306.996}
SPL {X  -159.990, Y  +429.021, Z    +0.000, E1   -63.228, E3 -241319.609}
SPL {X  -159.990, Y  +423.267, Z    +0.000, E1   -62.365, E3 -241331.907}
SPL {X  -159.990, Y  +418.218, Z    +0.000, E1   -61.769, E3 -241341.920}
SPL {X  -159.990, Y  +412.274, Z    +0.000, E1   -61.123, E3 -241353.324}
SPL {X  -159.990, Y  +408.631, Z    +0.000, E1   -60.233, E3 -241363.786}
SPL {X  -159.990, Y  +404.834, Z    +0.000, E1   -59.529, E3 -241373.241}
SPL {X  -159.990, Y  +397.866, Z    +0.000, E1   -58.924, E3 -241386.328}
SPL {X  -159.990, Y  +387.403, Z    +0.000, E1   -58.805, E3 -241400.424}
SPL {X  -159.948, Y  +378.844, Z    +0.000, E1   -58.798, E3 -241411.463}
SPL {X  -159.570, Y  +370.916, Z    +0.000, E1   -58.738, E3 -241422.059}
SPL {X  -158.865, Y  +363.563, Z    +0.000, E1   -58.615, E3 -241432.268}
SPL {X  -157.976, Y  +357.197, Z    +0.000, E1   -58.476, E3 -241441.369}
SPL {X  -156.730, Y  +350.368, Z    +0.000, E1   -58.276, E3 -241451.464}
SPL {X  -155.026, Y  +342.956, Z    +0.000, E1   -58.003, E3 -241462.737}
SPL {X  -152.946, Y  +335.551, Z    +0.000, E1   -57.653, E3 -241474.384}
SPL {X  -150.899, Y  +329.336, Z    +0.000, E1   -57.290, E3 -241484.450}
SPL {X  -149.179, Y  +324.687, Z    +0.000, E1   -56.983, E3 -241492.140}
SPL {X  -147.281, Y  +320.009, Z    +0.000, E1   -56.662, E3 -241499.966}
SPL {X  -144.114, Y  +313.017, Z    +0.000, E1   -56.131, E3 -241511.933}
SPL {X  -140.858, Y  +306.633, Z    +0.000, E1   -55.477, E3 -241523.228}
SPL {X  -138.338, Y  +302.130, Z    +0.000, E1   -54.992, E3 -241531.278}
SPL {X  -124.427, Y  +281.929, Z    +0.000, E1   -46.852, E3 -241635.514}
ENDSPLINE

SPLINE
SPL {X  -148.251, Y  +322.346, Z    +0.000, E1   -33.039, E3 -241723.439}
SPL {X  -157.534, Y  +354.574, Z    +0.000, E1   -18.815, E3 -241740.268}
SPL {X  -159.548, Y  +370.614, Z    +0.000, E1    -9.656, E3 -241743.894}
SPL {X  -159.928, Y  +378.035, Z    +0.000, E1    -4.866, E3 -241744.809}
SPL {X  -159.990, Y  +383.381, Z    +0.000, E1    -1.123, E3 -241745.130}
SPL {X  -159.990, Y  +386.348, Z    +0.000, E1    +1.571, E3 -241745.239}
SPL {X  -159.990, Y  +391.422, Z    +0.000, E1    +7.757, E3 -241745.613}
SPL {X  -159.990, Y  +396.843, Z    +0.000, E1   +15.720, E3 -241746.275}
SPL {X  -159.990, Y  +403.976, Z    +0.000, E1   +25.456, E3 -241747.813}
SPL {X  -159.990, Y  +417.120, Z    +0.000, E1   +39.678, E3 -241751.844}
SPL {X  -159.990, Y  +456.927, Z    +0.000, E1   +55.382, E3 -241773.704}
SPL {X  -159.990, Y  +530.047, Z    +0.000, E1   +58.901, E3 -241843.538}
SPL {X  -159.990, Y  +538.035, Z    +0.000, E1   +58.900, E3 -241853.764}
SPL {X  -159.990, Y  +546.883, Z    +0.000, E1   +58.912, E3 -241865.067}
SPL {X  -159.990, Y  +555.949, Z    +0.000, E1   +58.900, E3 -241876.687}
SPL {X  -159.990, Y  +563.718, Z    +0.000, E1   +58.903, E3 -241886.607}
SPL {X  -159.990, Y  +571.529, Z    +0.000, E1   +58.906, E3 -241896.591}
SPL {X  -159.990, Y  +579.859, Z    +0.000, E1   +58.907, E3 -241907.250}
SPL {X  -159.990, Y  +588.526, Z    +0.000, E1   +58.910, E3 -241918.324}
SPL {X  -159.990, Y  +596.521, Z    +0.000, E1   +58.902, E3 -241928.583}
SPL {X  -159.990, Y  +605.444, Z    +0.000, E1   +58.918, E3 -241939.973}
SPL {X  -159.990, Y  +618.101, Z    +0.000, E1   +58.946, E3 -241956.119}
SPL {X  -159.990, Y  +629.920, Z    +0.000, E1   +58.912, E3 -241971.312}
SPL {X  -159.990, Y  +642.398, Z    +0.000, E1   +58.947, E3 -241987.220}
SPL {X  -159.990, Y  +654.206, Z    +0.000, E1   +58.908, E3 -242002.391}
SPL {X  -159.990, Y  +661.562, Z    +0.000, E1   +58.900, E3 -242011.819}
SPL {X  -159.990, Y  +670.328, Z    +0.000, E1   +58.911, E3 -242023.018}
SPL {X  -159.795, Y  +679.404, Z    +0.000, E1   +58.876, E3 -242034.844}
SPL {X  -159.282, Y  +686.534, Z    +0.000, E1   +58.787, E3 -242044.517}
SPL {X  -158.463, Y  +693.553, Z    +0.000, E1   +58.665, E3 -242054.358}
SPL {X  -157.294, Y  +700.745, Z    +0.000, E1   +58.469, E3 -242064.809}
SPL {X  -156.031, Y  +706.871, Z    +0.000, E1   +58.260, E3 -242073.954}
SPL {X  -154.558, Y  +712.835, Z    +0.000, E1   +58.028, E3 -242083.081}
SPL {X  -152.750, Y  +719.085, Z    +0.000, E1   +57.721, E3 -242092.927}
SPL {X  -150.741, Y  +725.111, Z    +0.000, E1   +57.387, E3 -242102.632}
SPL {X  -148.665, Y  +730.623, Z    +0.000, E1   +57.007, E3 -242111.780}
SPL {X  -146.664, Y  +735.425, Z    +0.000, E1   +56.657, E3 -242119.870}
SPL {X  -143.496, Y  +742.251, Z    +0.000, E1   +56.124, E3 -242131.564}
SPL {X  -140.752, Y  +747.564, Z    +0.000, E1   +55.554, E3 -242140.971}
SPL {X  -138.492, Y  +751.605, Z    +0.000, E1   +55.137, E3 -242148.162}
SPL {X  -124.324, Y  +772.199, Z    +0.000, E1   +48.708, E3 -242227.170}
ENDSPLINE

SPLINE
SPL {X  -129.118, Y  +765.975, Z    +0.000, E1   +43.713, E3 -242291.655}
SPL {X  -146.252, Y  +736.362, Z    +0.000, E1   +34.795, E3 -242340.833}
SPL {X  -154.088, Y  +714.555, Z    +0.000, E1   +26.177, E3 -242354.850}
SPL {X  -156.688, Y  +703.837, Z    +0.000, E1   +21.096, E3 -242359.021}
SPL {X  -159.039, Y  +688.920, Z    +0.000, E1   +13.016, E3 -242362.953}
SPL {X  -159.888, Y  +677.224, Z    +0.000, E1    +5.773, E3 -242364.666}
SPL {X  -159.990, Y  +671.755, Z    +0.000, E1    +1.905, E3 -242365.069}
SPL {X  -159.990, Y  +668.898, Z    +0.000, E1    -0.346, E3 -242365.164}
SPL {X  -159.990, Y  +666.084, Z    +0.000, E1    -3.512, E3 -242365.286}
SPL {X  -159.990, Y  +662.904, Z    +0.000, E1    -7.618, E3 -242365.525}
SPL {X  -159.990, Y  +658.509, Z    +0.000, E1   -13.882, E3 -242366.061}
SPL {X  -159.990, Y  +652.317, Z    +0.000, E1   -22.778, E3 -242367.197}
SPL {X  -159.990, Y  +640.689, Z    +0.000, E1   -37.390, E3 -242368.739}
SPL {X  -159.990, Y  +585.634, Z    +0.000, E1   -68.681, E3 -242369.364}
SPL {X  -159.990, Y  +457.771, Z    +0.000, E1   -68.079, E3 -242459.925}
SPL {X  -159.990, Y  +453.218, Z    +0.000, E1   -67.322, E3 -242470.360}
SPL {X  -159.990, Y  +450.256, Z    +0.000, E1   -66.188, E3 -242482.293}
SPL {X  -159.990, Y  +445.667, Z    +0.000, E1   -65.356, E3 -242493.204}
SPL {X  -159.990, Y  +439.738, Z    +0.000, E1   -64.716, E3 -242504.017}
SPL {X  -159.990, Y  +435.528, Z    +0.000, E1   -63.972, E3 -242513.893}
SPL {X  -159.990, Y  +429.021, Z    +0.000, E1   -63.228, E3 -242526.506}
SPL {X  -159.990, Y  +423.267, Z    +0.000, E1   -62.365, E3 -242538.804}
SPL {X  -159.990, Y  +418.218, Z    +0.000, E1   -61.769, E3 -242548.816}
SPL {X  -159.990, Y  +412.274, Z    +0.000, E1   -61.123, E3 -242560.220}
SPL {X  -159.990, Y  +408.631, Z    +0.000, E1   -60.233, E3 -242570.683}
SPL {X  -159.990, Y  +404.834, Z    +0.000, E1   -59.529, E3 -242580.138}
SPL {X  -159.990, Y  +397.866, Z    +0.000, E1   -58.924, E3 -242593.225}
SPL {X  -159.990, Y  +387.403, Z    +0.000, E1   -58.805, E3 -242607.320}
SPL {X  -159.948, Y  +378.844, Z    +0.000, E1   -58.798, E3 -242618.360}
SPL {X  -159.570, Y  +370.916, Z    +0.000, E1   -58.738, E3 -242628.955}
SPL {X  -158.865, Y  +363.563, Z    +0.000, E1   -58.615, E3 -242639.165}
SPL {X  -157.976, Y  +357.197, Z    +0.000, E1   -58.476, E3 -242648.266}
SPL {X  -156.730, Y  +350.368, Z    +0.000, E1   -58.276, E3 -242658.361}
SPL {X  -155.026, Y  +342.956, Z    +0.000, E1   -58.003, E3 -242669.633}
SPL {X  -152.946, Y  +335.551, Z    +0.000, E1   -57.653, E3 -242681.281}
SPL {X  -150.105, Y  +327.135, Z    +0.000, E1   -57.196, E3 -242694.901}
SPL {X  -146.578, Y  +318.377, Z    +0.000, E1   -56.572, E3 -242709.594}
SPL {X  -143.463, Y  +311.683, Z    +0.000, E1   -55.972, E3 -242721.208}
SPL {X  -140.858, Y  +306.633, Z    +0.000, E1   -55.477, E3 -242730.125}
SPL {X  -138.338, Y  +302.130, Z    +0.000, E1   -54.992, E3 -242738.175}
SPL {X  -124.427, Y  +281.929, Z    +0.000, E1   -46.852, E3 -242842.411}
ENDSPLINE

SPLINE
SPL {X  -148.251, Y  +322.346, Z    +0.000, E1   -33.039, E3 -242930.336}
SPL {X  -156.481, Y  +349.177, Z    +0.000, E1   -21.514, E3 -242945.519}
SPL {X  -159.327, Y  +367.953, Z    +0.000, E1   -11.342, E3 -242950.310}
SPL {X  -159.973, Y  +380.173, Z    +0.000, E1    -3.469, E3 -242951.857}
SPL {X  -159.990, Y  +384.078, Z    +0.000, E1    -0.490, E3 -242952.055}
SPL {X  -159.990, Y  +386.348, Z    +0.000, E1    +1.571, E3 -242952.136}
SPL {X  -159.990, Y  +391.422, Z    +0.000, E1    +7.757, E3 -242952.510}
SPL {X  -159.990, Y  +399.099, Z    +0.000, E1   +18.787, E3 -242953.616}
SPL {X  -159.990, Y  +406.316, Z    +0.000, E1   +28.569, E3 -242955.294}
SPL {X  -159.990, Y  +417.120, Z    +0.000, E1   +39.678, E3 -242958.741}
SPL {X  -159.990, Y  +456.927, Z    +0.000, E1   +55.382, E3 -242980.601}
SPL {X  -159.990, Y  +530.047, Z    +0.000, E1   +58.901, E3 -243050.435}
SPL {X  -159.990, Y  +538.035, Z    +0.000, E1   +58.900, E3 -243060.660}
SPL {X  -159.990, Y  +546.883, Z    +0.000, E1   +58.912, E3 -243071.964}
SPL {X  -159.990, Y  +555.949, Z    +0.000, E1   +58.900, E3 -243083.583}
SPL {X  -159.990, Y  +563.718, Z    +0.000, E1   +58.903, E3 -243093.504}
SPL {X  -159.990, Y  +571.529, Z    +0.000, E1   +58.906, E3 -243103.488}
SPL {X  -159.990, Y  +579.859, Z    +0.000, E1   +58.907, E3 -243114.147}
SPL {X  -159.990, Y  +588.526, Z    +0.000, E1   +58.910, E3 -243125.221}
SPL {X  -159.990, Y  +596.521, Z    +0.000, E1   +58.902, E3 -243135.480}
SPL {X  -159.990, Y  +605.444, Z    +0.000, E1   +58.918, E3 -243146.869}
SPL {X  -159.990, Y  +618.101, Z    +0.000, E1   +58.946, E3 -243163.016}
SPL {X  -159.990, Y  +629.920, Z    +0.000, E1   +58.912, E3 -243178.209}
SPL {X  -159.990, Y  +638.424, Z    +0.000, E1   +58.901, E3 -243189.109}
SPL {X  -159.990, Y  +645.995, Z    +0.000, E1   +58.900, E3 -243198.797}
SPL {X  -159.990, Y  +654.206, Z    +0.000, E1   +58.908, E3 -243209.287}
SPL {X  -159.990, Y  +661.562, Z    +0.000, E1   +58.900, E3 -243218.716}
SPL {X  -159.990, Y  +670.328, Z    +0.000, E1   +58.911, E3 -243229.915}
SPL {X  -159.795, Y  +679.404, Z    +0.000, E1   +58.876, E3 -243241.740}
SPL {X  -159.282, Y  +686.534, Z    +0.000, E1   +58.787, E3 -243251.414}
SPL {X  -158.463, Y  +693.553, Z    +0.000, E1   +58.665, E3 -243261.255}
SPL {X  -157.294, Y  +700.745, Z    +0.000, E1   +58.469, E3 -243271.705}
SPL {X  -156.031, Y  +706.871, Z    +0.000, E1   +58.260, E3 -243280.851}
SPL {X  -154.558, Y  +712.835, Z    +0.000, E1   +58.028, E3 -243289.978}
SPL {X  -152.750, Y  +719.085, Z    +0.000, E1   +57.721, E3 -243299.824}
SPL {X  -150.741, Y  +725.111, Z    +0.000, E1   +57.387, E3 -243309.528}
SPL {X  -148.665, Y  +730.623, Z    +0.000, E1   +57.007, E3 -243318.677}
SPL {X  -146.664, Y  +735.425, Z    +0.000, E1   +56.657, E3 -243326.767}
SPL {X  -143.496, Y  +742.251, Z    +0.000, E1   +56.124, E3 -243338.460}
SPL {X  -140.752, Y  +747.564, Z    +0.000, E1   +55.554, E3 -243347.867}
SPL {X  -138.492, Y  +751.605, Z    +0.000, E1   +55.137, E3 -243355.059}
SPL {X  -124.324, Y  +772.199, Z    +0.000, E1   +48.708, E3 -243434.067}
ENDSPLINE

SPLINE
SPL {X  -129.118, Y  +765.975, Z    +0.000, E1   +43.713, E3 -243498.552}
SPL {X  -146.252, Y  +736.362, Z    +0.000, E1   +34.795, E3 -243547.730}
SPL {X  -155.916, Y  +707.374, Z    +0.000, E1   +22.878, E3 -243564.615}
SPL {X  -159.039, Y  +688.920, Z    +0.000, E1   +13.016, E3 -243569.850}
SPL {X  -159.777, Y  +679.762, Z    +0.000, E1    +7.372, E3 -243571.305}
SPL {X  -159.984, Y  +672.872, Z    +0.000, E1    +2.784, E3 -243571.902}
SPL {X  -159.990, Y  +669.598, Z    +0.000, E1    +0.205, E3 -243572.039}
SPL {X  -159.990, Y  +667.097, Z    +0.000, E1    -2.190, E3 -243572.134}
SPL {X  -159.990, Y  +662.904, Z    +0.000, E1    -7.618, E3 -243572.422}
SPL {X  -159.990, Y  +658.509, Z    +0.000, E1   -13.882, E3 -243572.958}
SPL {X  -159.990, Y  +652.317, Z    +0.000, E1   -22.778, E3 -243574.093}
SPL {X  -159.990, Y  +641.893, Z    +0.000, E1   -35.310, E3 -243577.058}
SPL {X  -159.990, Y  +636.123, Z    +0.000, E1   -46.139, E3 -243570.123}
SPL {X  -159.990, Y  +585.634, Z    +0.000, E1   -68.681, E3 -243576.260}
SPL {X  -159.990, Y  +457.771, Z    +0.000, E1   -68.079, E3 -243666.821}
SPL {X  -159.990, Y  +453.218, Z    +0.000, E1   -67.322, E3 -243677.257}
SPL {X  -159.990, Y  +450.256, Z    +0.000, E1   -66.188, E3 -243689.189}
SPL {X  -159.990, Y  +445.667, Z    +0.000, E1   -65.356, E3 -243700.101}
SPL {X  -159.990, Y  +439.738, Z    +0.000, E1   -64.716, E3 -243710.914}
SPL {X  -159.990, Y  +435.528, Z    +0.000, E1   -63.972, E3 -243720.789}
SPL {X  -159.990, Y  +429.021, Z    +0.000, E1   -63.228, E3 -243733.402}
SPL {X  -159.990, Y  +423.267, Z    +0.000, E1   -62.365, E3 -243745.700}
SPL {X  -159.990, Y  +418.218, Z    +0.000, E1   -61.769, E3 -243755.713}
SPL {X  -159.990, Y  +412.274, Z    +0.000, E1   -61.123, E3 -243767.117}
SPL {X  -159.990, Y  +408.631, Z    +0.000, E1   -60.233, E3 -243777.579}
SPL {X  -159.990, Y  +404.834, Z    +0.000, E1   -59.529, E3 -243787.034}
SPL {X  -159.990, Y  +397.866, Z    +0.000, E1   -58.924, E3 -243800.121}
SPL {X  -159.990, Y  +387.403, Z    +0.000, E1   -58.805, E3 -243814.217}
SPL {X  -159.948, Y  +378.844, Z    +0.000, E1   -58.798, E3 -243825.257}
SPL {X  -159.570, Y  +370.916, Z    +0.000, E1   -58.738, E3 -243835.852}
SPL {X  -158.865, Y  +363.563, Z    +0.000, E1   -58.615, E3 -243846.061}
SPL {X  -157.976, Y  +357.197, Z    +0.000, E1   -58.476, E3 -243855.162}
SPL {X  -156.730, Y  +350.368, Z    +0.000, E1   -58.276, E3 -243865.257}
SPL {X  -155.026, Y  +342.956, Z    +0.000, E1   -58.003, E3 -243876.530}
SPL {X  -152.946, Y  +335.551, Z    +0.000, E1   -57.653, E3 -243888.178}
SPL {X  -150.899, Y  +329.336, Z    +0.000, E1   -57.290, E3 -243898.243}
SPL {X  -149.179, Y  +324.687, Z    +0.000, E1   -56.983, E3 -243905.933}
SPL {X  -147.281, Y  +320.009, Z    +0.000, E1   -56.662, E3 -243913.759}
SPL {X  -144.114, Y  +313.017, Z    +0.000, E1   -56.131, E3 -243925.726}
SPL {X  -140.858, Y  +306.633, Z    +0.000, E1   -55.477, E3 -243937.022}
SPL {X  -138.338, Y  +302.130, Z    +0.000, E1   -54.992, E3 -243945.071}
SPL {X  -124.427, Y  +281.929, Z    +0.000, E1   -46.852, E3 -244049.307}
ENDSPLINE

SPLINE
SPL {X  -148.251, Y  +322.346, Z    +0.000, E1   -33.039, E3 -244137.232}
SPL {X  -157.534, Y  +354.574, Z    +0.000, E1   -18.815, E3 -244154.062}
SPL {X  -159.548, Y  +370.614, Z    +0.000, E1    -9.656, E3 -244157.687}
SPL {X  -159.928, Y  +378.035, Z    +0.000, E1    -4.866, E3 -244158.602}
SPL {X  -159.990, Y  +383.381, Z    +0.000, E1    -1.123, E3 -244158.923}
SPL {X  -159.990, Y  +386.348, Z    +0.000, E1    +1.571, E3 -244159.032}
SPL {X  -159.990, Y  +391.422, Z    +0.000, E1    +7.757, E3 -244159.406}
SPL {X  -159.990, Y  +396.843, Z    +0.000, E1   +15.720, E3 -244160.068}
SPL {X  -159.990, Y  +403.976, Z    +0.000, E1   +25.456, E3 -244161.606}
SPL {X  -159.990, Y  +417.120, Z    +0.000, E1   +39.678, E3 -244165.637}
SPL {X  -159.990, Y  +456.927, Z    +0.000, E1   +55.382, E3 -244187.498}
SPL {X  -159.990, Y  +530.047, Z    +0.000, E1   +58.901, E3 -244257.332}
SPL {X  -159.990, Y  +538.035, Z    +0.000, E1   +58.900, E3 -244267.557}
SPL {X  -159.990, Y  +546.883, Z    +0.000, E1   +58.912, E3 -244278.861}
SPL {X  -159.990, Y  +555.949, Z    +0.000, E1   +58.900, E3 -244290.480}
SPL {X  -159.990, Y  +563.718, Z    +0.000, E1   +58.903, E3 -244300.400}
SPL {X  -159.990, Y  +571.529, Z    +0.000, E1   +58.906, E3 -244310.384}
SPL {X  -159.990, Y  +579.859, Z    +0.000, E1   +58.907, E3 -244321.044}
SPL {X  -159.990, Y  +588.526, Z    +0.000, E1   +58.910, E3 -244332.117}
SPL {X  -159.990, Y  +596.521, Z    +0.000, E1   +58.902, E3 -244342.376}
SPL {X  -159.990, Y  +605.444, Z    +0.000, E1   +58.918, E3 -244353.766}
SPL {X  -159.990, Y  +618.101, Z    +0.000, E1   +58.946, E3 -244369.913}
SPL {X  -159.990, Y  +629.920, Z    +0.000, E1   +58.912, E3 -244385.105}
SPL {X  -159.990, Y  +642.398, Z    +0.000, E1   +58.947, E3 -244401.013}
SPL {X  -159.990, Y  +654.206, Z    +0.000, E1   +58.908, E3 -244416.184}
SPL {X  -159.990, Y  +661.562, Z    +0.000, E1   +58.900, E3 -244425.612}
SPL {X  -159.990, Y  +670.328, Z    +0.000, E1   +58.911, E3 -244436.811}
SPL {X  -159.795, Y  +679.404, Z    +0.000, E1   +58.876, E3 -244448.637}
SPL {X  -159.282, Y  +686.534, Z    +0.000, E1   +58.787, E3 -244458.310}
SPL {X  -158.463, Y  +693.553, Z    +0.000, E1   +58.665, E3 -244468.152}
SPL {X  -157.294, Y  +700.745, Z    +0.000, E1   +58.469, E3 -244478.602}
SPL {X  -156.031, Y  +706.871, Z    +0.000, E1   +58.260, E3 -244487.747}
SPL {X  -154.558, Y  +712.835, Z    +0.000, E1   +58.028, E3 -244496.874}
SPL {X  -152.750, Y  +719.085, Z    +0.000, E1   +57.721, E3 -244506.721}
SPL {X  -150.741, Y  +725.111, Z    +0.000, E1   +57.387, E3 -244516.425}
SPL {X  -148.665, Y  +730.623, Z    +0.000, E1   +57.007, E3 -244525.573}
SPL {X  -146.664, Y  +735.425, Z    +0.000, E1   +56.657, E3 -244533.663}
SPL {X  -143.496, Y  +742.251, Z    +0.000, E1   +56.124, E3 -244545.357}
SPL {X  -140.752, Y  +747.564, Z    +0.000, E1   +55.554, E3 -244554.764}
SPL {X  -138.492, Y  +751.605, Z    +0.000, E1   +55.137, E3 -244561.955}
SPL {X  -124.324, Y  +772.199, Z    +0.000, E1   +48.708, E3 -244640.963}
ENDSPLINE

SPLINE
SPL {X  -129.118, Y  +765.975, Z    +0.000, E1   +43.713, E3 -244705.449}
SPL {X  -146.252, Y  +736.362, Z    +0.000, E1   +34.795, E3 -244754.626}
SPL {X  -154.088, Y  +714.555, Z    +0.000, E1   +26.177, E3 -244768.643}
SPL {X  -156.688, Y  +703.837, Z    +0.000, E1   +21.096, E3 -244772.814}
SPL {X  -159.039, Y  +688.920, Z    +0.000, E1   +13.016, E3 -244776.746}
SPL {X  -159.888, Y  +677.224, Z    +0.000, E1    +5.773, E3 -244778.459}
SPL {X  -159.990, Y  +671.755, Z    +0.000, E1    +1.905, E3 -244778.863}
SPL {X  -159.990, Y  +668.898, Z    +0.000, E1    -0.346, E3 -244778.957}
SPL {X  -159.990, Y  +666.084, Z    +0.000, E1    -3.512, E3 -244779.079}
SPL {X  -159.990, Y  +662.904, Z    +0.000, E1    -7.618, E3 -244779.319}
SPL {X  -159.990, Y  +658.509, Z    +0.000, E1   -13.882, E3 -244779.854}
SPL {X  -159.990, Y  +652.317, Z    +0.000, E1   -22.778, E3 -244780.990}
SPL {X  -159.990, Y  +640.689, Z    +0.000, E1   -37.390, E3 -244782.532}
SPL {X  -159.990, Y  +585.634, Z    +0.000, E1   -68.681, E3 -244783.157}
SPL {X  -159.990, Y  +457.771, Z    +0.000, E1   -68.079, E3 -244873.718}
SPL {X  -159.990, Y  +453.218, Z    +0.000, E1   -67.322, E3 -244884.153}
SPL {X  -159.990, Y  +450.256, Z    +0.000, E1   -66.188, E3 -244896.086}
SPL {X  -159.990, Y  +445.667, Z    +0.000, E1   -65.356, E3 -244906.998}
SPL {X  -159.990, Y  +439.738, Z    +0.000, E1   -64.716, E3 -244917.810}
SPL {X  -159.990, Y  +435.528, Z    +0.000, E1   -63.972, E3 -244927.686}
SPL {X  -159.990, Y  +429.021, Z    +0.000, E1   -63.228, E3 -244940.299}
SPL {X  -159.990, Y  +423.267, Z    +0.000, E1   -62.365, E3 -244952.597}
SPL {X  -159.990, Y  +418.218, Z    +0.000, E1   -61.769, E3 -244962.609}
SPL {X  -159.990, Y  +412.274, Z    +0.000, E1   -61.123, E3 -244974.013}
SPL {X  -159.990, Y  +408.631, Z    +0.000, E1   -60.233, E3 -244984.476}
SPL {X  -159.990, Y  +404.834, Z    +0.000, E1   -59.529, E3 -244993.931}
SPL {X  -159.990, Y  +397.866, Z    +0.000, E1   -58.924, E3 -245007.018}
SPL {X  -159.990, Y  +387.403, Z    +0.000, E1   -58.805, E3 -245021.113}
SPL {X  -159.948, Y  +378.844, Z    +0.000, E1   -58.798, E3 -245032.153}
SPL {X  -159.570, Y  +370.916, Z    +0.000, E1   -58.738, E3 -245042.749}
SPL {X  -158.865, Y  +363.563, Z    +0.000, E1   -58.615, E3 -245052.958}
SPL {X  -157.976, Y  +357.197, Z    +0.000, E1   -58.476, E3 -245062.059}
SPL {X  -156.730, Y  +350.368, Z    +0.000, E1   -58.276, E3 -245072.154}
SPL {X  -155.026, Y  +342.956, Z    +0.000, E1   -58.003, E3 -245083.426}
SPL {X  -152.946, Y  +335.551, Z    +0.000, E1   -57.653, E3 -245095.074}
SPL {X  -150.105, Y  +327.135, Z    +0.000, E1   -57.196, E3 -245108.694}
SPL {X  -146.578, Y  +318.377, Z    +0.000, E1   -56.572, E3 -245123.387}
SPL {X  -143.463, Y  +311.683, Z    +0.000, E1   -55.972, E3 -245135.001}
SPL {X  -140.858, Y  +306.633, Z    +0.000, E1   -55.477, E3 -245143.918}
SPL {X  -138.338, Y  +302.130, Z    +0.000, E1   -54.992, E3 -245151.968}
SPL {X  -124.427, Y  +281.929, Z    +0.000, E1   -46.852, E3 -245256.204}
ENDSPLINE

SPLINE
SPL {X  -148.251, Y  +322.346, Z    +0.000, E1   -33.039, E3 -245344.129}
SPL {X  -156.481, Y  +349.177, Z    +0.000, E1   -21.514, E3 -245359.312}
SPL {X  -159.327, Y  +367.953, Z    +0.000, E1   -11.342, E3 -245364.103}
SPL {X  -159.973, Y  +380.173, Z    +0.000, E1    -3.469, E3 -245365.650}
SPL {X  -159.990, Y  +384.078, Z    +0.000, E1    -0.490, E3 -245365.848}
SPL {X  -159.990, Y  +386.348, Z    +0.000, E1    +1.571, E3 -245365.929}
SPL {X  -159.990, Y  +391.422, Z    +0.000, E1    +7.757, E3 -245366.303}
SPL {X  -159.990, Y  +399.099, Z    +0.000, E1   +18.787, E3 -245367.409}
SPL {X  -159.990, Y  +406.316, Z    +0.000, E1   +28.569, E3 -245369.087}
SPL {X  -159.990, Y  +417.120, Z    +0.000, E1   +39.678, E3 -245372.534}
SPL {X  -159.990, Y  +456.927, Z    +0.000, E1   +55.382, E3 -245394.394}
SPL {X  -159.990, Y  +530.047, Z    +0.000, E1   +58.901, E3 -245464.228}
SPL {X  -159.990, Y  +538.035, Z    +0.000, E1   +58.900, E3 -245474.453}
SPL {X  -159.990, Y  +546.883, Z    +0.000, E1   +58.912, E3 -245485.757}
SPL {X  -159.990, Y  +555.949, Z    +0.000, E1   +58.900, E3 -245497.377}
SPL {X  -159.990, Y  +563.718, Z    +0.000, E1   +58.903, E3 -245507.297}
SPL {X  -159.990, Y  +571.529, Z    +0.000, E1   +58.906, E3 -245517.281}
SPL {X  -159.990, Y  +579.859, Z    +0.000, E1   +58.907, E3 -245527.940}
SPL {X  -159.990, Y  +588.526, Z    +0.000, E1   +58.910, E3 -245539.014}
SPL {X  -159.990, Y  +596.521, Z    +0.000, E1   +58.902, E3 -245549.273}
SPL {X  -159.990, Y  +605.444, Z    +0.000, E1   +58.918, E3 -245560.662}
SPL {X  -159.990, Y  +618.101, Z    +0.000, E1   +58.946, E3 -245576.809}
SPL {X  -159.990, Y  +629.920, Z    +0.000, E1   +58.912, E3 -245592.002}
SPL {X  -159.990, Y  +638.424, Z    +0.000, E1   +58.901, E3 -245602.902}
SPL {X  -159.990, Y  +645.995, Z    +0.000, E1   +58.900, E3 -245612.590}
SPL {X  -159.990, Y  +654.206, Z    +0.000, E1   +58.908, E3 -245623.081}
SPL {X  -159.990, Y  +661.562, Z    +0.000, E1   +58.900, E3 -245632.509}
SPL {X  -159.990, Y  +670.328, Z    +0.000, E1   +58.911, E3 -245643.708}
SPL {X  -159.795, Y  +679.404, Z    +0.000, E1   +58.876, E3 -245655.533}
SPL {X  -159.282, Y  +686.534, Z    +0.000, E1   +58.787, E3 -245665.207}
SPL {X  -158.463, Y  +693.553, Z    +0.000, E1   +58.665, E3 -245675.048}
SPL {X  -157.294, Y  +700.745, Z    +0.000, E1   +58.469, E3 -245685.498}
SPL {X  -156.031, Y  +706.871, Z    +0.000, E1   +58.260, E3 -245694.644}
SPL {X  -154.558, Y  +712.835, Z    +0.000, E1   +58.028, E3 -245703.771}
SPL {X  -152.750, Y  +719.085, Z    +0.000, E1   +57.721, E3 -245713.617}
SPL {X  -150.741, Y  +725.111, Z    +0.000, E1   +57.387, E3 -245723.321}
SPL {X  -148.665, Y  +730.623, Z    +0.000, E1   +57.007, E3 -245732.470}
SPL {X  -146.664, Y  +735.425, Z    +0.000, E1   +56.657, E3 -245740.560}
SPL {X  -143.496, Y  +742.251, Z    +0.000, E1   +56.124, E3 -245752.253}
SPL {X  -140.752, Y  +747.564, Z    +0.000, E1   +55.554, E3 -245761.661}
SPL {X  -138.492, Y  +751.605, Z    +0.000, E1   +55.137, E3 -245768.852}
SPL {X  -124.324, Y  +772.199, Z    +0.000, E1   +48.708, E3 -245847.860}
ENDSPLINE

SPLINE
SPL {X  -129.118, Y  +765.975, Z    +0.000, E1   +43.713, E3 -245912.345}
SPL {X  -146.252, Y  +736.362, Z    +0.000, E1   +34.795, E3 -245961.523}
SPL {X  -154.088, Y  +714.555, Z    +0.000, E1   +26.177, E3 -245975.539}
SPL {X  -156.688, Y  +703.837, Z    +0.000, E1   +21.096, E3 -245979.711}
SPL {X  -159.039, Y  +688.920, Z    +0.000, E1   +13.016, E3 -245983.643}
SPL {X  -159.888, Y  +677.224, Z    +0.000, E1    +5.773, E3 -245985.356}
SPL {X  -159.990, Y  +670.275, Z    +0.000, E1    +0.854, E3 -245985.809}
SPL {X  -159.990, Y  +667.097, Z    +0.000, E1    -2.190, E3 -245985.927}
SPL {X  -159.990, Y  +662.904, Z    +0.000, E1    -7.618, E3 -245986.215}
SPL {X  -159.990, Y  +658.509, Z    +0.000, E1   -13.882, E3 -245986.751}
SPL {X  -159.990, Y  +652.317, Z    +0.000, E1   -22.778, E3 -245987.886}
SPL {X  -159.990, Y  +640.689, Z    +0.000, E1   -37.390, E3 -245989.429}
SPL {X  -159.990, Y  +585.634, Z    +0.000, E1   -68.681, E3 -245990.053}
SPL {X  -159.990, Y  +457.771, Z    +0.000, E1   -68.079, E3 -246080.614}
SPL {X  -159.990, Y  +453.218, Z    +0.000, E1   -67.322, E3 -246091.050}
SPL {X  -159.990, Y  +450.256, Z    +0.000, E1   -66.188, E3 -246102.982}
SPL {X  -159.990, Y  +445.667, Z    +0.000, E1   -65.356, E3 -246113.894}
SPL {X  -159.990, Y  +439.738, Z    +0.000, E1   -64.716, E3 -246124.707}
SPL {X  -159.990, Y  +435.528, Z    +0.000, E1   -63.972, E3 -246134.583}
SPL {X  -159.990, Y  +429.021, Z    +0.000, E1   -63.228, E3 -246147.195}
SPL {X  -159.990, Y  +423.267, Z    +0.000, E1   -62.365, E3 -246159.493}
SPL {X  -159.990, Y  +418.218, Z    +0.000, E1   -61.769, E3 -246169.506}
SPL {X  -159.990, Y  +412.274, Z    +0.000, E1   -61.123, E3 -246180.910}
SPL {X  -159.990, Y  +408.631, Z    +0.000, E1   -60.233, E3 -246191.372}
SPL {X  -159.990, Y  +404.834, Z    +0.000, E1   -59.529, E3 -246200.827}
SPL {X  -159.990, Y  +397.866, Z    +0.000, E1   -58.924, E3 -246213.915}
SPL {X  -159.990, Y  +387.403, Z    +0.000, E1   -58.805, E3 -246228.010}
SPL {X  -159.948, Y  +378.844, Z    +0.000, E1   -58.798, E3 -246239.050}
SPL {X  -159.570, Y  +370.916, Z    +0.000, E1   -58.738, E3 -246249.645}
SPL {X  -158.865, Y  +363.563, Z    +0.000, E1   -58.615, E3 -246259.855}
SPL {X  -157.976, Y  +357.197, Z    +0.000, E1   -58.476, E3 -246268.955}
SPL {X  -156.730, Y  +350.368, Z    +0.000, E1   -58.276, E3 -246279.051}
SPL {X  -155.026, Y  +342.956, Z    +0.000, E1   -58.003, E3 -246290.323}
SPL {X  -152.946, Y  +335.551, Z    +0.000, E1   -57.653, E3 -246301.971}
SPL {X  -150.899, Y  +329.336, Z    +0.000, E1   -57.290, E3 -246312.036}
SPL {X  -149.179, Y  +324.687, Z    +0.000, E1   -56.983, E3 -246319.726}
SPL {X  -146.578, Y  +318.377, Z    +0.000, E1   -56.572, E3 -246330.284}
SPL {X  -143.463, Y  +311.683, Z    +0.000, E1   -55.972, E3 -246341.897}
SPL {X  -140.858, Y  +306.633, Z    +0.000, E1   -55.477, E3 -246350.815}
SPL {X  -138.338, Y  +302.130, Z    +0.000, E1   -54.992, E3 -246358.864}
SPL {X  -124.427, Y  +281.929, Z    +0.000, E1   -46.852, E3 -246463.100}
ENDSPLINE

SPLINE
SPL {X  -138.506, Y  +302.419, Z    +0.000, E1   -39.451, E3 -246529.075}
SPL {X  -149.686, Y  +326.013, Z    +0.000, E1   -31.658, E3 -246554.211}
SPL {X  -156.481, Y  +349.177, Z    +0.000, E1   -21.514, E3 -246566.209}
SPL {X  -159.327, Y  +367.953, Z    +0.000, E1   -11.342, E3 -246571.000}
SPL {X  -159.973, Y  +380.173, Z    +0.000, E1    -3.469, E3 -246572.547}
SPL {X  -159.990, Y  +384.078, Z    +0.000, E1    -0.490, E3 -246572.745}
SPL {X  -159.990, Y  +385.440, Z    +0.000, E1    +0.747, E3 -246572.785}
SPL {X  -159.990, Y  +388.179, Z    +0.000, E1    +3.660, E3 -246572.926}
SPL {X  -159.990, Y  +394.222, Z    +0.000, E1   +11.674, E3 -246573.519}
SPL {X  -159.990, Y  +403.976, Z    +0.000, E1   +25.456, E3 -246575.399}
SPL {X  -159.990, Y  +417.120, Z    +0.000, E1   +39.678, E3 -246579.430}
SPL {X  -159.990, Y  +456.927, Z    +0.000, E1   +55.382, E3 -246601.291}
SPL {X  -159.990, Y  +530.047, Z    +0.000, E1   +58.901, E3 -246671.125}
SPL {X  -159.990, Y  +538.035, Z    +0.000, E1   +58.900, E3 -246681.350}
SPL {X  -159.990, Y  +546.883, Z    +0.000, E1   +58.912, E3 -246692.654}
SPL {X  -159.990, Y  +555.949, Z    +0.000, E1   +58.900, E3 -246704.273}
SPL {X  -159.990, Y  +563.718, Z    +0.000, E1   +58.903, E3 -246714.193}
SPL {X  -159.990, Y  +571.529, Z    +0.000, E1   +58.906, E3 -246724.177}
SPL {X  -159.990, Y  +579.859, Z    +0.000, E1   +58.907, E3 -246734.837}
SPL {X  -159.990, Y  +588.526, Z    +0.000, E1   +58.910, E3 -246745.910}
SPL {X  -159.990, Y  +596.521, Z    +0.000, E1   +58.902, E3 -246756.169}
SPL {X  -159.990, Y  +605.444, Z    +0.000, E1   +58.918, E3 -246767.559}
SPL {X  -159.990, Y  +613.908, Z    +0.000, E1   +58.900, E3 -246778.418}
SPL {X  -159.990, Y  +621.342, Z    +0.000, E1   +58.904, E3 -246787.926}
SPL {X  -159.990, Y  +629.920, Z    +0.000, E1   +58.912, E3 -246798.899}
SPL {X  -159.990, Y  +642.398, Z    +0.000, E1   +58.947, E3 -246814.806}
SPL {X  -159.990, Y  +654.206, Z    +0.000, E1   +58.908, E3 -246829.977}
SPL {X  -159.990, Y  +661.562, Z    +0.000, E1   +58.900, E3 -246839.405}
SPL {X  -159.990, Y  +670.328, Z    +0.000, E1   +58.911, E3 -246850.605}
SPL {X  -159.795, Y  +679.404, Z    +0.000, E1   +58.876, E3 -246862.430}
SPL {X  -159.282, Y  +686.534, Z    +0.000, E1   +58.787, E3 -246872.104}
SPL {X  -158.463, Y  +693.553, Z    +0.000, E1   +58.665, E3 -246881.945}
SPL {X  -157.294, Y  +700.745, Z    +0.000, E1   +58.469, E3 -246892.395}
SPL {X  -156.031, Y  +706.871, Z    +0.000, E1   +58.260, E3 -246901.540}
SPL {X  -154.558, Y  +712.835, Z    +0.000, E1   +58.028, E3 -246910.668}
SPL {X  -152.750, Y  +719.085, Z    +0.000, E1   +57.721, E3 -246920.514}
SPL {X  -150.741, Y  +725.111, Z    +0.000, E1   +57.387, E3 -246930.218}
SPL {X  -148.665, Y  +730.623, Z    +0.000, E1   +57.007, E3 -246939.366}
SPL {X  -146.664, Y  +735.425, Z    +0.000, E1   +56.657, E3 -246947.457}
SPL {X  -143.496, Y  +742.251, Z    +0.000, E1   +56.124, E3 -246959.150}
SPL {X  -140.752, Y  +747.564, Z    +0.000, E1   +55.554, E3 -246968.557}
SPL {X  -138.492, Y  +751.605, Z    +0.000, E1   +55.137, E3 -246975.748}
SPL {X  -124.324, Y  +772.199, Z    +0.000, E1   +48.708, E3 -247054.756}
ENDSPLINE

SPLINE
SPL {X  -129.118, Y  +765.975, Z    +0.000, E1   +43.713, E3 -247119.242}
SPL {X  -146.252, Y  +736.362, Z    +0.000, E1   +34.795, E3 -247168.419}
SPL {X  -154.088, Y  +714.555, Z    +0.000, E1   +26.177, E3 -247182.436}
SPL {X  -156.688, Y  +703.837, Z    +0.000, E1   +21.096, E3 -247186.607}
SPL {X  -159.039, Y  +688.920, Z    +0.000, E1   +13.016, E3 -247190.539}
SPL {X  -159.888, Y  +677.224, Z    +0.000, E1    +5.773, E3 -247192.252}
SPL {X  -159.990, Y  +671.755, Z    +0.000, E1    +1.905, E3 -247192.656}
SPL {X  -159.990, Y  +669.598, Z    +0.000, E1    +0.205, E3 -247192.729}
SPL {X  -159.990, Y  +667.097, Z    +0.000, E1    -2.190, E3 -247192.824}
SPL {X  -159.990, Y  +662.904, Z    +0.000, E1    -7.618, E3 -247193.112}
SPL {X  -159.990, Y  +658.509, Z    +0.000, E1   -13.882, E3 -247193.647}
SPL {X  -159.990, Y  +652.317, Z    +0.000, E1   -22.778, E3 -247194.783}
SPL {X  -159.990, Y  +641.893, Z    +0.000, E1   -35.310, E3 -247197.748}
SPL {X  -159.990, Y  +636.123, Z    +0.000, E1   -46.139, E3 -247190.813}
SPL {X  -159.990, Y  +585.634, Z    +0.000, E1   -68.681, E3 -247196.950}
SPL {X  -159.990, Y  +457.771, Z    +0.000, E1   -68.079, E3 -247287.511}
SPL {X  -159.990, Y  +453.218, Z    +0.000, E1   -67.322, E3 -247297.946}
SPL {X  -159.990, Y  +450.256, Z    +0.000, E1   -66.188, E3 -247309.879}
SPL {X  -159.990, Y  +445.667, Z    +0.000, E1   -65.356, E3 -247320.791}
SPL {X  -159.990, Y  +439.738, Z    +0.000, E1   -64.716, E3 -247331.603}
SPL {X  -159.990, Y  +435.528, Z    +0.000, E1   -63.972, E3 -247341.479}
SPL {X  -159.990, Y  +429.021, Z    +0.000, E1   -63.228, E3 -247354.092}
SPL {X  -159.990, Y  +423.267, Z    +0.000, E1   -62.365, E3 -247366.390}
SPL {X  -159.990, Y  +418.218, Z    +0.000, E1   -61.769, E3 -247376.402}
SPL {X  -159.990, Y  +412.274, Z    +0.000, E1   -61.123, E3 -247387.806}
SPL {X  -159.990, Y  +408.631, Z    +0.000, E1   -60.233, E3 -247398.269}
SPL {X  -159.990, Y  +404.834, Z    +0.000, E1   -59.529, E3 -247407.724}
SPL {X  -159.990, Y  +397.866, Z    +0.000, E1   -58.924, E3 -247420.811}
SPL {X  -159.990, Y  +387.403, Z    +0.000, E1   -58.805, E3 -247434.906}
SPL {X  -159.948, Y  +378.844, Z    +0.000, E1   -58.798, E3 -247445.946}
SPL {X  -159.570, Y  +370.916, Z    +0.000, E1   -58.738, E3 -247456.542}
SPL {X  -158.865, Y  +363.563, Z    +0.000, E1   -58.615, E3 -247466.751}
SPL {X  -157.976, Y  +357.197, Z    +0.000, E1   -58.476, E3 -247475.852}
SPL {X  -156.730, Y  +350.368, Z    +0.000, E1   -58.276, E3 -247485.947}
SPL {X  -155.026, Y  +342.956, Z    +0.000, E1   -58.003, E3 -247497.219}
SPL {X  -152.946, Y  +335.551, Z    +0.000, E1   -57.653, E3 -247508.867}
SPL {X  -150.899, Y  +329.336, Z    +0.000, E1   -57.290, E3 -247518.933}
SPL {X  -149.179, Y  +324.687, Z    +0.000, E1   -56.983, E3 -247526.622}
SPL {X  -147.281, Y  +320.009, Z    +0.000, E1   -56.662, E3 -247534.448}
SPL {X  -144.114, Y  +313.017, Z    +0.000, E1   -56.131, E3 -247546.416}
SPL {X  -140.858, Y  +306.633, Z    +0.000, E1   -55.477, E3 -247557.711}
SPL {X  -138.338, Y  +302.130, Z    +0.000, E1   -54.992, E3 -247565.761}
SPL {X  -124.427, Y  +281.929, Z    +0.000, E1   -46.852, E3 -247669.997}
ENDSPLINE

SPLINE
SPL {X  -148.251, Y  +322.346, Z    +0.000, E1   -33.039, E3 -247757.922}
SPL {X  -157.534, Y  +354.574, Z    +0.000, E1   -18.815, E3 -247774.751}
SPL {X  -159.548, Y  +370.614, Z    +0.000, E1    -9.656, E3 -247778.377}
SPL {X  -159.928, Y  +378.035, Z    +0.000, E1    -4.866, E3 -247779.292}
SPL {X  -159.990, Y  +383.381, Z    +0.000, E1    -1.123, E3 -247779.613}
SPL {X  -159.990, Y  +386.348, Z    +0.000, E1    +1.571, E3 -247779.722}
SPL {X  -159.990, Y  +391.422, Z    +0.000, E1    +7.757, E3 -247780.096}
SPL {X  -159.990, Y  +396.843, Z    +0.000, E1   +15.720, E3 -247780.758}
SPL {X  -159.990, Y  +403.976, Z    +0.000, E1   +25.456, E3 -247782.296}
SPL {X  -159.990, Y  +417.120, Z    +0.000, E1   +39.678, E3 -247786.327}
SPL {X  -159.990, Y  +456.927, Z    +0.000, E1   +55.382, E3 -247808.187}
SPL {X  -159.990, Y  +530.047, Z    +0.000, E1   +58.901, E3 -247878.021}
SPL {X  -159.990, Y  +538.035, Z    +0.000, E1   +58.900, E3 -247888.247}
SPL {X  -159.990, Y  +546.883, Z    +0.000, E1   +58.912, E3 -247899.550}
SPL {X  -159.990, Y  +555.949, Z    +0.000, E1   +58.900, E3 -247911.170}
SPL {X  -159.990, Y  +563.718, Z    +0.000, E1   +58.903, E3 -247921.090}
SPL {X  -159.990, Y  +571.529, Z    +0.000, E1   +58.906, E3 -247931.074}
SPL {X  -159.990, Y  +579.859, Z    +0.000, E1   +58.907, E3 -247941.733}
SPL {X  -159.990, Y  +588.526, Z    +0.000, E1   +58.910, E3 -247952.807}
SPL {X  -159.990, Y  +596.521, Z    +0.000, E1   +58.902, E3 -247963.066}
SPL {X  -159.990, Y  +605.444, Z    +0.000, E1   +58.918, E3 -247974.455}
SPL {X  -159.990, Y  +613.908, Z    +0.000, E1   +58.900, E3 -247985.315}
SPL {X  -159.990, Y  +621.342, Z    +0.000, E1   +58.904, E3 -247994.823}
SPL {X  -159.990, Y  +629.920, Z    +0.000, E1   +58.912, E3 -248005.795}
SPL {X  -159.990, Y  +642.398, Z    +0.000, E1   +58.947, E3 -248021.703}
SPL {X  -159.990, Y  +654.206, Z    +0.000, E1   +58.908, E3 -248036.874}
SPL {X  -159.990, Y  +661.562, Z    +0.000, E1   +58.900, E3 -248046.302}
SPL {X  -159.990, Y  +670.328, Z    +0.000, E1   +58.911, E3 -248057.501}
SPL {X  -159.795, Y  +679.404, Z    +0.000, E1   +58.876, E3 -248069.326}
SPL {X  -159.282, Y  +686.534, Z    +0.000, E1   +58.787, E3 -248079.000}
SPL {X  -158.463, Y  +693.553, Z    +0.000, E1   +58.665, E3 -248088.841}
SPL {X  -157.294, Y  +700.745, Z    +0.000, E1   +58.469, E3 -248099.291}
SPL {X  -156.031, Y  +706.871, Z    +0.000, E1   +58.260, E3 -248108.437}
SPL {X  -154.558, Y  +712.835, Z    +0.000, E1   +58.028, E3 -248117.564}
SPL {X  -152.750, Y  +719.085, Z    +0.000, E1   +57.721, E3 -248127.410}
SPL {X  -150.741, Y  +725.111, Z    +0.000, E1   +57.387, E3 -248137.114}
SPL {X  -148.665, Y  +730.623, Z    +0.000, E1   +57.007, E3 -248146.263}
SPL {X  -146.664, Y  +735.425, Z    +0.000, E1   +56.657, E3 -248154.353}
SPL {X  -144.631, Y  +739.900, Z    +0.000, E1   +56.280, E3 -248162.039}
SPL {X  -141.795, Y  +745.600, Z    +0.000, E1   +55.801, E3 -248171.921}
SPL {X  -138.492, Y  +751.605, Z    +0.000, E1   +55.137, E3 -248182.645}
SPL {X  -124.324, Y  +772.199, Z    +0.000, E1   +48.708, E3 -248261.653}
ENDSPLINE

